eRFID[71].nCardNumber;eRFID[71].bROPPPuttedChecked;	eRFID[71].bROPPPutted;		eRFID[71].bROPPCapped;		eRFID[71].bROPPCappingAborted;eRFID[71].bROPPCappingOK; eRFID[71].bROPPCappingChecked;eRFID[71].bFormPresent; eRFID[71].bBottlePresent; eRFID[71].bDosingTwoPhases; eRFID[71].nDispencerNr; eRFID[71].nDispencerNrSecondPhase; eRFID[71].lrDoseVolumeSV; eRFID[71].lrDoseVolumeCV; eRFID[71].lrDoseVolumeSVSecondPhase; eRFID[71].lrDoseVolumeCVSecondPhase; eRFID[71].bDosed;	eRFID[71].bDoseAborted; eRFID[71].bWeighed; eRFID[71].lrWeightSV; eRFID[71].lrWeightCV; eRFID[71].lrWeightMeasuredCV; eRFID[71].bWeightOK; eRFID[71].bCapPutted; eRFID[71].bCapChecked; eRFID[71].bCapOK; eRFID[71].bCapGripperScrewed; eRFID[71].bCapGripperScrewAborted; eRFID[71].bBottleTransferedToExit; eRFID[71].bBottleTransferedToLabeler; eRFID[71].lrWeightDif; eRFID[71].lrMinWeightCV;eRFID[71].lrMaxWeightCV;
eRFID[72].nCardNumber;eRFID[72].bROPPPuttedChecked;	eRFID[72].bROPPPutted;		eRFID[72].bROPPCapped;		eRFID[72].bROPPCappingAborted;eRFID[72].bROPPCappingOK; eRFID[72].bROPPCappingChecked;eRFID[72].bFormPresent; eRFID[72].bBottlePresent; eRFID[72].bDosingTwoPhases; eRFID[72].nDispencerNr; eRFID[72].nDispencerNrSecondPhase; eRFID[72].lrDoseVolumeSV; eRFID[72].lrDoseVolumeCV; eRFID[72].lrDoseVolumeSVSecondPhase; eRFID[72].lrDoseVolumeCVSecondPhase; eRFID[72].bDosed;	eRFID[72].bDoseAborted; eRFID[72].bWeighed; eRFID[72].lrWeightSV; eRFID[72].lrWeightCV; eRFID[72].lrWeightMeasuredCV; eRFID[72].bWeightOK; eRFID[72].bCapPutted; eRFID[72].bCapChecked; eRFID[72].bCapOK; eRFID[72].bCapGripperScrewed; eRFID[72].bCapGripperScrewAborted; eRFID[72].bBottleTransferedToExit; eRFID[72].bBottleTransferedToLabeler; eRFID[72].lrWeightDif; eRFID[72].lrMinWeightCV;eRFID[72].lrMaxWeightCV;
eRFID[73].nCardNumber;eRFID[73].bROPPPuttedChecked;	eRFID[73].bROPPPutted;		eRFID[73].bROPPCapped;		eRFID[73].bROPPCappingAborted;eRFID[73].bROPPCappingOK; eRFID[73].bROPPCappingChecked;eRFID[73].bFormPresent; eRFID[73].bBottlePresent; eRFID[73].bDosingTwoPhases; eRFID[73].nDispencerNr; eRFID[73].nDispencerNrSecondPhase; eRFID[73].lrDoseVolumeSV; eRFID[73].lrDoseVolumeCV; eRFID[73].lrDoseVolumeSVSecondPhase; eRFID[73].lrDoseVolumeCVSecondPhase; eRFID[73].bDosed;	eRFID[73].bDoseAborted; eRFID[73].bWeighed; eRFID[73].lrWeightSV; eRFID[73].lrWeightCV; eRFID[73].lrWeightMeasuredCV; eRFID[73].bWeightOK; eRFID[73].bCapPutted; eRFID[73].bCapChecked; eRFID[73].bCapOK; eRFID[73].bCapGripperScrewed; eRFID[73].bCapGripperScrewAborted; eRFID[73].bBottleTransferedToExit; eRFID[73].bBottleTransferedToLabeler; eRFID[73].lrWeightDif; eRFID[73].lrMinWeightCV;eRFID[73].lrMaxWeightCV;
eRFID[74].nCardNumber;eRFID[74].bROPPPuttedChecked;	eRFID[74].bROPPPutted;		eRFID[74].bROPPCapped;		eRFID[74].bROPPCappingAborted;eRFID[74].bROPPCappingOK; eRFID[74].bROPPCappingChecked;eRFID[74].bFormPresent; eRFID[74].bBottlePresent; eRFID[74].bDosingTwoPhases; eRFID[74].nDispencerNr; eRFID[74].nDispencerNrSecondPhase; eRFID[74].lrDoseVolumeSV; eRFID[74].lrDoseVolumeCV; eRFID[74].lrDoseVolumeSVSecondPhase; eRFID[74].lrDoseVolumeCVSecondPhase; eRFID[74].bDosed;	eRFID[74].bDoseAborted; eRFID[74].bWeighed; eRFID[74].lrWeightSV; eRFID[74].lrWeightCV; eRFID[74].lrWeightMeasuredCV; eRFID[74].bWeightOK; eRFID[74].bCapPutted; eRFID[74].bCapChecked; eRFID[74].bCapOK; eRFID[74].bCapGripperScrewed; eRFID[74].bCapGripperScrewAborted; eRFID[74].bBottleTransferedToExit; eRFID[74].bBottleTransferedToLabeler; eRFID[74].lrWeightDif; eRFID[74].lrMinWeightCV;eRFID[74].lrMaxWeightCV;
eRFID[75].nCardNumber;eRFID[75].bROPPPuttedChecked;	eRFID[75].bROPPPutted;		eRFID[75].bROPPCapped;		eRFID[75].bROPPCappingAborted;eRFID[75].bROPPCappingOK; eRFID[75].bROPPCappingChecked;eRFID[75].bFormPresent; eRFID[75].bBottlePresent; eRFID[75].bDosingTwoPhases; eRFID[75].nDispencerNr; eRFID[75].nDispencerNrSecondPhase; eRFID[75].lrDoseVolumeSV; eRFID[75].lrDoseVolumeCV; eRFID[75].lrDoseVolumeSVSecondPhase; eRFID[75].lrDoseVolumeCVSecondPhase; eRFID[75].bDosed;	eRFID[75].bDoseAborted; eRFID[75].bWeighed; eRFID[75].lrWeightSV; eRFID[75].lrWeightCV; eRFID[75].lrWeightMeasuredCV; eRFID[75].bWeightOK; eRFID[75].bCapPutted; eRFID[75].bCapChecked; eRFID[75].bCapOK; eRFID[75].bCapGripperScrewed; eRFID[75].bCapGripperScrewAborted; eRFID[75].bBottleTransferedToExit; eRFID[75].bBottleTransferedToLabeler; eRFID[75].lrWeightDif; eRFID[75].lrMinWeightCV;eRFID[75].lrMaxWeightCV;
eRFID[76].nCardNumber;eRFID[76].bROPPPuttedChecked;	eRFID[76].bROPPPutted;		eRFID[76].bROPPCapped;		eRFID[76].bROPPCappingAborted;eRFID[76].bROPPCappingOK; eRFID[76].bROPPCappingChecked;eRFID[76].bFormPresent; eRFID[76].bBottlePresent; eRFID[76].bDosingTwoPhases; eRFID[76].nDispencerNr; eRFID[76].nDispencerNrSecondPhase; eRFID[76].lrDoseVolumeSV; eRFID[76].lrDoseVolumeCV; eRFID[76].lrDoseVolumeSVSecondPhase; eRFID[76].lrDoseVolumeCVSecondPhase; eRFID[76].bDosed;	eRFID[76].bDoseAborted; eRFID[76].bWeighed; eRFID[76].lrWeightSV; eRFID[76].lrWeightCV; eRFID[76].lrWeightMeasuredCV; eRFID[76].bWeightOK; eRFID[76].bCapPutted; eRFID[76].bCapChecked; eRFID[76].bCapOK; eRFID[76].bCapGripperScrewed; eRFID[76].bCapGripperScrewAborted; eRFID[76].bBottleTransferedToExit; eRFID[76].bBottleTransferedToLabeler; eRFID[76].lrWeightDif; eRFID[76].lrMinWeightCV;eRFID[76].lrMaxWeightCV;
eRFID[77].nCardNumber;eRFID[77].bROPPPuttedChecked;	eRFID[77].bROPPPutted;		eRFID[77].bROPPCapped;		eRFID[77].bROPPCappingAborted;eRFID[77].bROPPCappingOK; eRFID[77].bROPPCappingChecked;eRFID[77].bFormPresent; eRFID[77].bBottlePresent; eRFID[77].bDosingTwoPhases; eRFID[77].nDispencerNr; eRFID[77].nDispencerNrSecondPhase; eRFID[77].lrDoseVolumeSV; eRFID[77].lrDoseVolumeCV; eRFID[77].lrDoseVolumeSVSecondPhase; eRFID[77].lrDoseVolumeCVSecondPhase; eRFID[77].bDosed;	eRFID[77].bDoseAborted; eRFID[77].bWeighed; eRFID[77].lrWeightSV; eRFID[77].lrWeightCV; eRFID[77].lrWeightMeasuredCV; eRFID[77].bWeightOK; eRFID[77].bCapPutted; eRFID[77].bCapChecked; eRFID[77].bCapOK; eRFID[77].bCapGripperScrewed; eRFID[77].bCapGripperScrewAborted; eRFID[77].bBottleTransferedToExit; eRFID[77].bBottleTransferedToLabeler; eRFID[77].lrWeightDif; eRFID[77].lrMinWeightCV;eRFID[77].lrMaxWeightCV;
eRFID[78].nCardNumber;eRFID[78].bROPPPuttedChecked;	eRFID[78].bROPPPutted;		eRFID[78].bROPPCapped;		eRFID[78].bROPPCappingAborted;eRFID[78].bROPPCappingOK; eRFID[78].bROPPCappingChecked;eRFID[78].bFormPresent; eRFID[78].bBottlePresent; eRFID[78].bDosingTwoPhases; eRFID[78].nDispencerNr; eRFID[78].nDispencerNrSecondPhase; eRFID[78].lrDoseVolumeSV; eRFID[78].lrDoseVolumeCV; eRFID[78].lrDoseVolumeSVSecondPhase; eRFID[78].lrDoseVolumeCVSecondPhase; eRFID[78].bDosed;	eRFID[78].bDoseAborted; eRFID[78].bWeighed; eRFID[78].lrWeightSV; eRFID[78].lrWeightCV; eRFID[78].lrWeightMeasuredCV; eRFID[78].bWeightOK; eRFID[78].bCapPutted; eRFID[78].bCapChecked; eRFID[78].bCapOK; eRFID[78].bCapGripperScrewed; eRFID[78].bCapGripperScrewAborted; eRFID[78].bBottleTransferedToExit; eRFID[78].bBottleTransferedToLabeler; eRFID[78].lrWeightDif; eRFID[78].lrMinWeightCV;eRFID[78].lrMaxWeightCV;
eRFID[79].nCardNumber;eRFID[79].bROPPPuttedChecked;	eRFID[79].bROPPPutted;		eRFID[79].bROPPCapped;		eRFID[79].bROPPCappingAborted;eRFID[79].bROPPCappingOK; eRFID[79].bROPPCappingChecked;eRFID[79].bFormPresent; eRFID[79].bBottlePresent; eRFID[79].bDosingTwoPhases; eRFID[79].nDispencerNr; eRFID[79].nDispencerNrSecondPhase; eRFID[79].lrDoseVolumeSV; eRFID[79].lrDoseVolumeCV; eRFID[79].lrDoseVolumeSVSecondPhase; eRFID[79].lrDoseVolumeCVSecondPhase; eRFID[79].bDosed;	eRFID[79].bDoseAborted; eRFID[79].bWeighed; eRFID[79].lrWeightSV; eRFID[79].lrWeightCV; eRFID[79].lrWeightMeasuredCV; eRFID[79].bWeightOK; eRFID[79].bCapPutted; eRFID[79].bCapChecked; eRFID[79].bCapOK; eRFID[79].bCapGripperScrewed; eRFID[79].bCapGripperScrewAborted; eRFID[79].bBottleTransferedToExit; eRFID[79].bBottleTransferedToLabeler; eRFID[79].lrWeightDif; eRFID[79].lrMinWeightCV;eRFID[79].lrMaxWeightCV;
eRFID[80].nCardNumber;eRFID[80].bROPPPuttedChecked;	eRFID[80].bROPPPutted;		eRFID[80].bROPPCapped;		eRFID[80].bROPPCappingAborted;eRFID[80].bROPPCappingOK; eRFID[80].bROPPCappingChecked;eRFID[80].bFormPresent; eRFID[80].bBottlePresent; eRFID[80].bDosingTwoPhases; eRFID[80].nDispencerNr; eRFID[80].nDispencerNrSecondPhase; eRFID[80].lrDoseVolumeSV; eRFID[80].lrDoseVolumeCV; eRFID[80].lrDoseVolumeSVSecondPhase; eRFID[80].lrDoseVolumeCVSecondPhase; eRFID[80].bDosed;	eRFID[80].bDoseAborted; eRFID[80].bWeighed; eRFID[80].lrWeightSV; eRFID[80].lrWeightCV; eRFID[80].lrWeightMeasuredCV; eRFID[80].bWeightOK; eRFID[80].bCapPutted; eRFID[80].bCapChecked; eRFID[80].bCapOK; eRFID[80].bCapGripperScrewed; eRFID[80].bCapGripperScrewAborted; eRFID[80].bBottleTransferedToExit; eRFID[80].bBottleTransferedToLabeler; eRFID[80].lrWeightDif; eRFID[80].lrMinWeightCV;eRFID[80].lrMaxWeightCV;
eRFID[81].nCardNumber;eRFID[81].bROPPPuttedChecked;	eRFID[81].bROPPPutted;		eRFID[81].bROPPCapped;		eRFID[81].bROPPCappingAborted;eRFID[81].bROPPCappingOK; eRFID[81].bROPPCappingChecked;eRFID[81].bFormPresent; eRFID[81].bBottlePresent; eRFID[81].bDosingTwoPhases; eRFID[81].nDispencerNr; eRFID[81].nDispencerNrSecondPhase; eRFID[81].lrDoseVolumeSV; eRFID[81].lrDoseVolumeCV; eRFID[81].lrDoseVolumeSVSecondPhase; eRFID[81].lrDoseVolumeCVSecondPhase; eRFID[81].bDosed;	eRFID[81].bDoseAborted; eRFID[81].bWeighed; eRFID[81].lrWeightSV; eRFID[81].lrWeightCV; eRFID[81].lrWeightMeasuredCV; eRFID[81].bWeightOK; eRFID[81].bCapPutted; eRFID[81].bCapChecked; eRFID[81].bCapOK; eRFID[81].bCapGripperScrewed; eRFID[81].bCapGripperScrewAborted; eRFID[81].bBottleTransferedToExit; eRFID[81].bBottleTransferedToLabeler; eRFID[81].lrWeightDif; eRFID[81].lrMinWeightCV;eRFID[81].lrMaxWeightCV;
eRFID[82].nCardNumber;eRFID[82].bROPPPuttedChecked;	eRFID[82].bROPPPutted;		eRFID[82].bROPPCapped;		eRFID[82].bROPPCappingAborted;eRFID[82].bROPPCappingOK; eRFID[82].bROPPCappingChecked;eRFID[82].bFormPresent; eRFID[82].bBottlePresent; eRFID[82].bDosingTwoPhases; eRFID[82].nDispencerNr; eRFID[82].nDispencerNrSecondPhase; eRFID[82].lrDoseVolumeSV; eRFID[82].lrDoseVolumeCV; eRFID[82].lrDoseVolumeSVSecondPhase; eRFID[82].lrDoseVolumeCVSecondPhase; eRFID[82].bDosed;	eRFID[82].bDoseAborted; eRFID[82].bWeighed; eRFID[82].lrWeightSV; eRFID[82].lrWeightCV; eRFID[82].lrWeightMeasuredCV; eRFID[82].bWeightOK; eRFID[82].bCapPutted; eRFID[82].bCapChecked; eRFID[82].bCapOK; eRFID[82].bCapGripperScrewed; eRFID[82].bCapGripperScrewAborted; eRFID[82].bBottleTransferedToExit; eRFID[82].bBottleTransferedToLabeler; eRFID[82].lrWeightDif; eRFID[82].lrMinWeightCV;eRFID[82].lrMaxWeightCV;
eRFID[83].nCardNumber;eRFID[83].bROPPPuttedChecked;	eRFID[83].bROPPPutted;		eRFID[83].bROPPCapped;		eRFID[83].bROPPCappingAborted;eRFID[83].bROPPCappingOK; eRFID[83].bROPPCappingChecked;eRFID[83].bFormPresent; eRFID[83].bBottlePresent; eRFID[83].bDosingTwoPhases; eRFID[83].nDispencerNr; eRFID[83].nDispencerNrSecondPhase; eRFID[83].lrDoseVolumeSV; eRFID[83].lrDoseVolumeCV; eRFID[83].lrDoseVolumeSVSecondPhase; eRFID[83].lrDoseVolumeCVSecondPhase; eRFID[83].bDosed;	eRFID[83].bDoseAborted; eRFID[83].bWeighed; eRFID[83].lrWeightSV; eRFID[83].lrWeightCV; eRFID[83].lrWeightMeasuredCV; eRFID[83].bWeightOK; eRFID[83].bCapPutted; eRFID[83].bCapChecked; eRFID[83].bCapOK; eRFID[83].bCapGripperScrewed; eRFID[83].bCapGripperScrewAborted; eRFID[83].bBottleTransferedToExit; eRFID[83].bBottleTransferedToLabeler; eRFID[83].lrWeightDif; eRFID[83].lrMinWeightCV;eRFID[83].lrMaxWeightCV;
eRFID[84].nCardNumber;eRFID[84].bROPPPuttedChecked;	eRFID[84].bROPPPutted;		eRFID[84].bROPPCapped;		eRFID[84].bROPPCappingAborted;eRFID[84].bROPPCappingOK; eRFID[84].bROPPCappingChecked;eRFID[84].bFormPresent; eRFID[84].bBottlePresent; eRFID[84].bDosingTwoPhases; eRFID[84].nDispencerNr; eRFID[84].nDispencerNrSecondPhase; eRFID[84].lrDoseVolumeSV; eRFID[84].lrDoseVolumeCV; eRFID[84].lrDoseVolumeSVSecondPhase; eRFID[84].lrDoseVolumeCVSecondPhase; eRFID[84].bDosed;	eRFID[84].bDoseAborted; eRFID[84].bWeighed; eRFID[84].lrWeightSV; eRFID[84].lrWeightCV; eRFID[84].lrWeightMeasuredCV; eRFID[84].bWeightOK; eRFID[84].bCapPutted; eRFID[84].bCapChecked; eRFID[84].bCapOK; eRFID[84].bCapGripperScrewed; eRFID[84].bCapGripperScrewAborted; eRFID[84].bBottleTransferedToExit; eRFID[84].bBottleTransferedToLabeler; eRFID[84].lrWeightDif; eRFID[84].lrMinWeightCV;eRFID[84].lrMaxWeightCV;
eRFID[85].nCardNumber;eRFID[85].bROPPPuttedChecked;	eRFID[85].bROPPPutted;		eRFID[85].bROPPCapped;		eRFID[85].bROPPCappingAborted;eRFID[85].bROPPCappingOK; eRFID[85].bROPPCappingChecked;eRFID[85].bFormPresent; eRFID[85].bBottlePresent; eRFID[85].bDosingTwoPhases; eRFID[85].nDispencerNr; eRFID[85].nDispencerNrSecondPhase; eRFID[85].lrDoseVolumeSV; eRFID[85].lrDoseVolumeCV; eRFID[85].lrDoseVolumeSVSecondPhase; eRFID[85].lrDoseVolumeCVSecondPhase; eRFID[85].bDosed;	eRFID[85].bDoseAborted; eRFID[85].bWeighed; eRFID[85].lrWeightSV; eRFID[85].lrWeightCV; eRFID[85].lrWeightMeasuredCV; eRFID[85].bWeightOK; eRFID[85].bCapPutted; eRFID[85].bCapChecked; eRFID[85].bCapOK; eRFID[85].bCapGripperScrewed; eRFID[85].bCapGripperScrewAborted; eRFID[85].bBottleTransferedToExit; eRFID[85].bBottleTransferedToLabeler; eRFID[85].lrWeightDif; eRFID[85].lrMinWeightCV;eRFID[85].lrMaxWeightCV;
eRFID[86].nCardNumber;eRFID[86].bROPPPuttedChecked;	eRFID[86].bROPPPutted;		eRFID[86].bROPPCapped;		eRFID[86].bROPPCappingAborted;eRFID[86].bROPPCappingOK; eRFID[86].bROPPCappingChecked;eRFID[86].bFormPresent; eRFID[86].bBottlePresent; eRFID[86].bDosingTwoPhases; eRFID[86].nDispencerNr; eRFID[86].nDispencerNrSecondPhase; eRFID[86].lrDoseVolumeSV; eRFID[86].lrDoseVolumeCV; eRFID[86].lrDoseVolumeSVSecondPhase; eRFID[86].lrDoseVolumeCVSecondPhase; eRFID[86].bDosed;	eRFID[86].bDoseAborted; eRFID[86].bWeighed; eRFID[86].lrWeightSV; eRFID[86].lrWeightCV; eRFID[86].lrWeightMeasuredCV; eRFID[86].bWeightOK; eRFID[86].bCapPutted; eRFID[86].bCapChecked; eRFID[86].bCapOK; eRFID[86].bCapGripperScrewed; eRFID[86].bCapGripperScrewAborted; eRFID[86].bBottleTransferedToExit; eRFID[86].bBottleTransferedToLabeler; eRFID[86].lrWeightDif; eRFID[86].lrMinWeightCV;eRFID[86].lrMaxWeightCV;
eRFID[87].nCardNumber;eRFID[87].bROPPPuttedChecked;	eRFID[87].bROPPPutted;		eRFID[87].bROPPCapped;		eRFID[87].bROPPCappingAborted;eRFID[87].bROPPCappingOK; eRFID[87].bROPPCappingChecked;eRFID[87].bFormPresent; eRFID[87].bBottlePresent; eRFID[87].bDosingTwoPhases; eRFID[87].nDispencerNr; eRFID[87].nDispencerNrSecondPhase; eRFID[87].lrDoseVolumeSV; eRFID[87].lrDoseVolumeCV; eRFID[87].lrDoseVolumeSVSecondPhase; eRFID[87].lrDoseVolumeCVSecondPhase; eRFID[87].bDosed;	eRFID[87].bDoseAborted; eRFID[87].bWeighed; eRFID[87].lrWeightSV; eRFID[87].lrWeightCV; eRFID[87].lrWeightMeasuredCV; eRFID[87].bWeightOK; eRFID[87].bCapPutted; eRFID[87].bCapChecked; eRFID[87].bCapOK; eRFID[87].bCapGripperScrewed; eRFID[87].bCapGripperScrewAborted; eRFID[87].bBottleTransferedToExit; eRFID[87].bBottleTransferedToLabeler; eRFID[87].lrWeightDif; eRFID[87].lrMinWeightCV;eRFID[87].lrMaxWeightCV;
eRFID[88].nCardNumber;eRFID[88].bROPPPuttedChecked;	eRFID[88].bROPPPutted;		eRFID[88].bROPPCapped;		eRFID[88].bROPPCappingAborted;eRFID[88].bROPPCappingOK; eRFID[88].bROPPCappingChecked;eRFID[88].bFormPresent; eRFID[88].bBottlePresent; eRFID[88].bDosingTwoPhases; eRFID[88].nDispencerNr; eRFID[88].nDispencerNrSecondPhase; eRFID[88].lrDoseVolumeSV; eRFID[88].lrDoseVolumeCV; eRFID[88].lrDoseVolumeSVSecondPhase; eRFID[88].lrDoseVolumeCVSecondPhase; eRFID[88].bDosed;	eRFID[88].bDoseAborted; eRFID[88].bWeighed; eRFID[88].lrWeightSV; eRFID[88].lrWeightCV; eRFID[88].lrWeightMeasuredCV; eRFID[88].bWeightOK; eRFID[88].bCapPutted; eRFID[88].bCapChecked; eRFID[88].bCapOK; eRFID[88].bCapGripperScrewed; eRFID[88].bCapGripperScrewAborted; eRFID[88].bBottleTransferedToExit; eRFID[88].bBottleTransferedToLabeler; eRFID[88].lrWeightDif; eRFID[88].lrMinWeightCV;eRFID[88].lrMaxWeightCV;
eRFID[89].nCardNumber;eRFID[89].bROPPPuttedChecked;	eRFID[89].bROPPPutted;		eRFID[89].bROPPCapped;		eRFID[89].bROPPCappingAborted;eRFID[89].bROPPCappingOK; eRFID[89].bROPPCappingChecked;eRFID[89].bFormPresent; eRFID[89].bBottlePresent; eRFID[89].bDosingTwoPhases; eRFID[89].nDispencerNr; eRFID[89].nDispencerNrSecondPhase; eRFID[89].lrDoseVolumeSV; eRFID[89].lrDoseVolumeCV; eRFID[89].lrDoseVolumeSVSecondPhase; eRFID[89].lrDoseVolumeCVSecondPhase; eRFID[89].bDosed;	eRFID[89].bDoseAborted; eRFID[89].bWeighed; eRFID[89].lrWeightSV; eRFID[89].lrWeightCV; eRFID[89].lrWeightMeasuredCV; eRFID[89].bWeightOK; eRFID[89].bCapPutted; eRFID[89].bCapChecked; eRFID[89].bCapOK; eRFID[89].bCapGripperScrewed; eRFID[89].bCapGripperScrewAborted; eRFID[89].bBottleTransferedToExit; eRFID[89].bBottleTransferedToLabeler; eRFID[89].lrWeightDif; eRFID[89].lrMinWeightCV;eRFID[89].lrMaxWeightCV;
eRFID[90].nCardNumber;eRFID[90].bROPPPuttedChecked;	eRFID[90].bROPPPutted;		eRFID[90].bROPPCapped;		eRFID[90].bROPPCappingAborted;eRFID[90].bROPPCappingOK; eRFID[90].bROPPCappingChecked;eRFID[90].bFormPresent; eRFID[90].bBottlePresent; eRFID[90].bDosingTwoPhases; eRFID[90].nDispencerNr; eRFID[90].nDispencerNrSecondPhase; eRFID[90].lrDoseVolumeSV; eRFID[90].lrDoseVolumeCV; eRFID[90].lrDoseVolumeSVSecondPhase; eRFID[90].lrDoseVolumeCVSecondPhase; eRFID[90].bDosed;	eRFID[90].bDoseAborted; eRFID[90].bWeighed; eRFID[90].lrWeightSV; eRFID[90].lrWeightCV; eRFID[90].lrWeightMeasuredCV; eRFID[90].bWeightOK; eRFID[90].bCapPutted; eRFID[90].bCapChecked; eRFID[90].bCapOK; eRFID[90].bCapGripperScrewed; eRFID[90].bCapGripperScrewAborted; eRFID[90].bBottleTransferedToExit; eRFID[90].bBottleTransferedToLabeler; eRFID[90].lrWeightDif; eRFID[90].lrMinWeightCV;eRFID[90].lrMaxWeightCV;
eRFID[91].nCardNumber;eRFID[91].bROPPPuttedChecked;	eRFID[91].bROPPPutted;		eRFID[91].bROPPCapped;		eRFID[91].bROPPCappingAborted;eRFID[91].bROPPCappingOK; eRFID[91].bROPPCappingChecked;eRFID[91].bFormPresent; eRFID[91].bBottlePresent; eRFID[91].bDosingTwoPhases; eRFID[91].nDispencerNr; eRFID[91].nDispencerNrSecondPhase; eRFID[91].lrDoseVolumeSV; eRFID[91].lrDoseVolumeCV; eRFID[91].lrDoseVolumeSVSecondPhase; eRFID[91].lrDoseVolumeCVSecondPhase; eRFID[91].bDosed;	eRFID[91].bDoseAborted; eRFID[91].bWeighed; eRFID[91].lrWeightSV; eRFID[91].lrWeightCV; eRFID[91].lrWeightMeasuredCV; eRFID[91].bWeightOK; eRFID[91].bCapPutted; eRFID[91].bCapChecked; eRFID[91].bCapOK; eRFID[91].bCapGripperScrewed; eRFID[91].bCapGripperScrewAborted; eRFID[91].bBottleTransferedToExit; eRFID[91].bBottleTransferedToLabeler; eRFID[91].lrWeightDif; eRFID[91].lrMinWeightCV;eRFID[91].lrMaxWeightCV;
eRFID[92].nCardNumber;eRFID[92].bROPPPuttedChecked;	eRFID[92].bROPPPutted;		eRFID[92].bROPPCapped;		eRFID[92].bROPPCappingAborted;eRFID[92].bROPPCappingOK; eRFID[92].bROPPCappingChecked;eRFID[92].bFormPresent; eRFID[92].bBottlePresent; eRFID[92].bDosingTwoPhases; eRFID[92].nDispencerNr; eRFID[92].nDispencerNrSecondPhase; eRFID[92].lrDoseVolumeSV; eRFID[92].lrDoseVolumeCV; eRFID[92].lrDoseVolumeSVSecondPhase; eRFID[92].lrDoseVolumeCVSecondPhase; eRFID[92].bDosed;	eRFID[92].bDoseAborted; eRFID[92].bWeighed; eRFID[92].lrWeightSV; eRFID[92].lrWeightCV; eRFID[92].lrWeightMeasuredCV; eRFID[92].bWeightOK; eRFID[92].bCapPutted; eRFID[92].bCapChecked; eRFID[92].bCapOK; eRFID[92].bCapGripperScrewed; eRFID[92].bCapGripperScrewAborted; eRFID[92].bBottleTransferedToExit; eRFID[92].bBottleTransferedToLabeler; eRFID[92].lrWeightDif; eRFID[92].lrMinWeightCV;eRFID[92].lrMaxWeightCV;
eRFID[93].nCardNumber;eRFID[93].bROPPPuttedChecked;	eRFID[93].bROPPPutted;		eRFID[93].bROPPCapped;		eRFID[93].bROPPCappingAborted;eRFID[93].bROPPCappingOK; eRFID[93].bROPPCappingChecked;eRFID[93].bFormPresent; eRFID[93].bBottlePresent; eRFID[93].bDosingTwoPhases; eRFID[93].nDispencerNr; eRFID[93].nDispencerNrSecondPhase; eRFID[93].lrDoseVolumeSV; eRFID[93].lrDoseVolumeCV; eRFID[93].lrDoseVolumeSVSecondPhase; eRFID[93].lrDoseVolumeCVSecondPhase; eRFID[93].bDosed;	eRFID[93].bDoseAborted; eRFID[93].bWeighed; eRFID[93].lrWeightSV; eRFID[93].lrWeightCV; eRFID[93].lrWeightMeasuredCV; eRFID[93].bWeightOK; eRFID[93].bCapPutted; eRFID[93].bCapChecked; eRFID[93].bCapOK; eRFID[93].bCapGripperScrewed; eRFID[93].bCapGripperScrewAborted; eRFID[93].bBottleTransferedToExit; eRFID[93].bBottleTransferedToLabeler; eRFID[93].lrWeightDif; eRFID[93].lrMinWeightCV;eRFID[93].lrMaxWeightCV;
eRFID[94].nCardNumber;eRFID[94].bROPPPuttedChecked;	eRFID[94].bROPPPutted;		eRFID[94].bROPPCapped;		eRFID[94].bROPPCappingAborted;eRFID[94].bROPPCappingOK; eRFID[94].bROPPCappingChecked;eRFID[94].bFormPresent; eRFID[94].bBottlePresent; eRFID[94].bDosingTwoPhases; eRFID[94].nDispencerNr; eRFID[94].nDispencerNrSecondPhase; eRFID[94].lrDoseVolumeSV; eRFID[94].lrDoseVolumeCV; eRFID[94].lrDoseVolumeSVSecondPhase; eRFID[94].lrDoseVolumeCVSecondPhase; eRFID[94].bDosed;	eRFID[94].bDoseAborted; eRFID[94].bWeighed; eRFID[94].lrWeightSV; eRFID[94].lrWeightCV; eRFID[94].lrWeightMeasuredCV; eRFID[94].bWeightOK; eRFID[94].bCapPutted; eRFID[94].bCapChecked; eRFID[94].bCapOK; eRFID[94].bCapGripperScrewed; eRFID[94].bCapGripperScrewAborted; eRFID[94].bBottleTransferedToExit; eRFID[94].bBottleTransferedToLabeler; eRFID[94].lrWeightDif; eRFID[94].lrMinWeightCV;eRFID[94].lrMaxWeightCV;
eRFID[95].nCardNumber;eRFID[95].bROPPPuttedChecked;	eRFID[95].bROPPPutted;		eRFID[95].bROPPCapped;		eRFID[95].bROPPCappingAborted;eRFID[95].bROPPCappingOK; eRFID[95].bROPPCappingChecked;eRFID[95].bFormPresent; eRFID[95].bBottlePresent; eRFID[95].bDosingTwoPhases; eRFID[95].nDispencerNr; eRFID[95].nDispencerNrSecondPhase; eRFID[95].lrDoseVolumeSV; eRFID[95].lrDoseVolumeCV; eRFID[95].lrDoseVolumeSVSecondPhase; eRFID[95].lrDoseVolumeCVSecondPhase; eRFID[95].bDosed;	eRFID[95].bDoseAborted; eRFID[95].bWeighed; eRFID[95].lrWeightSV; eRFID[95].lrWeightCV; eRFID[95].lrWeightMeasuredCV; eRFID[95].bWeightOK; eRFID[95].bCapPutted; eRFID[95].bCapChecked; eRFID[95].bCapOK; eRFID[95].bCapGripperScrewed; eRFID[95].bCapGripperScrewAborted; eRFID[95].bBottleTransferedToExit; eRFID[95].bBottleTransferedToLabeler; eRFID[95].lrWeightDif; eRFID[95].lrMinWeightCV;eRFID[95].lrMaxWeightCV;
eRFID[96].nCardNumber;eRFID[96].bROPPPuttedChecked;	eRFID[96].bROPPPutted;		eRFID[96].bROPPCapped;		eRFID[96].bROPPCappingAborted;eRFID[96].bROPPCappingOK; eRFID[96].bROPPCappingChecked;eRFID[96].bFormPresent; eRFID[96].bBottlePresent; eRFID[96].bDosingTwoPhases; eRFID[96].nDispencerNr; eRFID[96].nDispencerNrSecondPhase; eRFID[96].lrDoseVolumeSV; eRFID[96].lrDoseVolumeCV; eRFID[96].lrDoseVolumeSVSecondPhase; eRFID[96].lrDoseVolumeCVSecondPhase; eRFID[96].bDosed;	eRFID[96].bDoseAborted; eRFID[96].bWeighed; eRFID[96].lrWeightSV; eRFID[96].lrWeightCV; eRFID[96].lrWeightMeasuredCV; eRFID[96].bWeightOK; eRFID[96].bCapPutted; eRFID[96].bCapChecked; eRFID[96].bCapOK; eRFID[96].bCapGripperScrewed; eRFID[96].bCapGripperScrewAborted; eRFID[96].bBottleTransferedToExit; eRFID[96].bBottleTransferedToLabeler; eRFID[96].lrWeightDif; eRFID[96].lrMinWeightCV;eRFID[96].lrMaxWeightCV;
eRFID[97].nCardNumber;eRFID[97].bROPPPuttedChecked;	eRFID[97].bROPPPutted;		eRFID[97].bROPPCapped;		eRFID[97].bROPPCappingAborted;eRFID[97].bROPPCappingOK; eRFID[97].bROPPCappingChecked;eRFID[97].bFormPresent; eRFID[97].bBottlePresent; eRFID[97].bDosingTwoPhases; eRFID[97].nDispencerNr; eRFID[97].nDispencerNrSecondPhase; eRFID[97].lrDoseVolumeSV; eRFID[97].lrDoseVolumeCV; eRFID[97].lrDoseVolumeSVSecondPhase; eRFID[97].lrDoseVolumeCVSecondPhase; eRFID[97].bDosed;	eRFID[97].bDoseAborted; eRFID[97].bWeighed; eRFID[97].lrWeightSV; eRFID[97].lrWeightCV; eRFID[97].lrWeightMeasuredCV; eRFID[97].bWeightOK; eRFID[97].bCapPutted; eRFID[97].bCapChecked; eRFID[97].bCapOK; eRFID[97].bCapGripperScrewed; eRFID[97].bCapGripperScrewAborted; eRFID[97].bBottleTransferedToExit; eRFID[97].bBottleTransferedToLabeler; eRFID[97].lrWeightDif; eRFID[97].lrMinWeightCV;eRFID[97].lrMaxWeightCV;
eRFID[98].nCardNumber;eRFID[98].bROPPPuttedChecked;	eRFID[98].bROPPPutted;		eRFID[98].bROPPCapped;		eRFID[98].bROPPCappingAborted;eRFID[98].bROPPCappingOK; eRFID[98].bROPPCappingChecked;eRFID[98].bFormPresent; eRFID[98].bBottlePresent; eRFID[98].bDosingTwoPhases; eRFID[98].nDispencerNr; eRFID[98].nDispencerNrSecondPhase; eRFID[98].lrDoseVolumeSV; eRFID[98].lrDoseVolumeCV; eRFID[98].lrDoseVolumeSVSecondPhase; eRFID[98].lrDoseVolumeCVSecondPhase; eRFID[98].bDosed;	eRFID[98].bDoseAborted; eRFID[98].bWeighed; eRFID[98].lrWeightSV; eRFID[98].lrWeightCV; eRFID[98].lrWeightMeasuredCV; eRFID[98].bWeightOK; eRFID[98].bCapPutted; eRFID[98].bCapChecked; eRFID[98].bCapOK; eRFID[98].bCapGripperScrewed; eRFID[98].bCapGripperScrewAborted; eRFID[98].bBottleTransferedToExit; eRFID[98].bBottleTransferedToLabeler; eRFID[98].lrWeightDif; eRFID[98].lrMinWeightCV;eRFID[98].lrMaxWeightCV;
eRFID[99].nCardNumber;eRFID[99].bROPPPuttedChecked;	eRFID[99].bROPPPutted;		eRFID[99].bROPPCapped;		eRFID[99].bROPPCappingAborted;eRFID[99].bROPPCappingOK; eRFID[99].bROPPCappingChecked;eRFID[99].bFormPresent; eRFID[99].bBottlePresent; eRFID[99].bDosingTwoPhases; eRFID[99].nDispencerNr; eRFID[99].nDispencerNrSecondPhase; eRFID[99].lrDoseVolumeSV; eRFID[99].lrDoseVolumeCV; eRFID[99].lrDoseVolumeSVSecondPhase; eRFID[99].lrDoseVolumeCVSecondPhase; eRFID[99].bDosed;	eRFID[99].bDoseAborted; eRFID[99].bWeighed; eRFID[99].lrWeightSV; eRFID[99].lrWeightCV; eRFID[99].lrWeightMeasuredCV; eRFID[99].bWeightOK; eRFID[99].bCapPutted; eRFID[99].bCapChecked; eRFID[99].bCapOK; eRFID[99].bCapGripperScrewed; eRFID[99].bCapGripperScrewAborted; eRFID[99].bBottleTransferedToExit; eRFID[99].bBottleTransferedToLabeler; eRFID[99].lrWeightDif; eRFID[99].lrMinWeightCV;eRFID[99].lrMaxWeightCV;
eRFID[100].nCardNumber;eRFID[100].bROPPPuttedChecked;eRFID[100].bROPPPutted;	eRFID[100].bROPPCapped;		eRFID[100].bROPPCappingAborted;eRFID[100].bROPPCappingOK;eRFID[100].bROPPCappingChecked;;eRFID[100].bFormPresent; eRFID[100].bBottlePresent; eRFID[100].bDosingTwoPhases; eRFID[100].nDispencerNr; eRFID[100].nDispencerNrSecondPhase; eRFID[100].lrDoseVolumeSV; eRFID[100].lrDoseVolumeCV; eRFID[100].lrDoseVolumeSVSecondPhase; eRFID[100].lrDoseVolumeCVSecondPhase; eRFID[100].bDoseAborted; eRFID[100].bWeighed; eRFID[100].lrWeightSV; eRFID[100].lrWeightCV; eRFID[100].lrWeightMeasuredCV; eRFID[100].bWeightOK; eRFID[100].bCapPutted; eRFID[100].bCapChecked; eRFID[100].bCapOK; eRFID[100].bCapGripperScrewed; eRFID[100].bCapGripperScrewAborted; eRFID[100].bBottleTransferedToExit; eRFID[100].bBottleTransferedToLabeler; eRFID[100].lrWeightDif; eRFID[100].lrMinWeightCV;eRFID[100].lrMinWeightCV;;
END_ACTION

ACTION aWizard:


VIS.bCapPuttedCheckSensor :=P09_CapPuttedCheck.IbCapPuttedCheckSensor;
VIS.bCapCorrectCheckCapOnSensor	:=P11_CapCorrectCheck.IbCapCorrectCheckCapOKSensor;
VIS.bCapCorrectCheckCapNotScrewedSensor :=P11_CapCorrectCheck.IbCapCorrectCheckCapNotScrewedSensor;
END_ACTION

METHOD FormDescription : STRING
VAR_INPUT
	B:BOOL;
	W:BOOL;
	N:BOOL;
	Z:BOOL;
END_VAR
IF Z THEN
	FormDescription := 'Z';
ELSIF N THEN
	FormDescription := 'N';
ELSIF W THEN
	FormDescription := 'W';
ELSIF B THEN
	FormDescription := 'B';
ELSE
	FormDescription := '';
END_IF
END_METHOD

END_PROGRAM

// ---- POUs/FB/FB_ReasonBadPackage.TcPOU
(*
Nazwa:			FB_ReasonBadPackage
Opis:			Powód odrzuceń 
Wersja:			v0.1
Data:			2019-12-17
Autor:			DP
Urzadzenia:		
Konfiguracja:	
Info: 
- 
*)
FUNCTION_BLOCK FB_ReasonBadPackage
VAR_INPUT
	bEnable: BOOL;				//Zezwolenie na pracę
	bReset:BOOL;				//Stop awaryjny nieaktywny
	tTime:TIME;					//
	bAddReason:BOOL;			//Dodaj pomiar
	bReason1:BOOL;
	sReason1Description:STRING;	//Nazwa stacji nr 1
	bReason2:BOOL;
	sReason2Description:STRING;	//Nazwa stacji nr 2
	bReason3:BOOL;
	sReason3Description:STRING;	//Nazwa stacji nr 3
	bReason4:BOOL;
	sReason4Description:STRING;	//Nazwa stacji nr 4
	bReason5:BOOL;
	sReason5Description:STRING;	//Nazwa stacji nr 5
	bReason6:BOOL;
	sReason6Description:STRING;	//Nazwa stacji nr 6
	bReason7:BOOL;
	sReason7Description:STRING;	//Nazwa stacji nr 7
	bReason8:BOOL;
	sReason8Description:STRING;	//Nazwa stacji nr 8
	bReason9:BOOL;
	sReason9Description:STRING;	//Nazwa stacji nr 9
	bReason10:BOOL;
	sReason10Description:STRING;	//Nazwa stacji nr 10
	bReason11:BOOL;
	sReason11Description:STRING;	//Nazwa stacji nr 10
	bReason12:BOOL;
	sReason12Description:STRING;	//Nazwa stacji nr 10
END_VAR

VAR_OUTPUT
	sBadPackage1:STRING;		//Opis powodu odrzuceń nr 1
	sBadPackage2:STRING;		//Opis powodu odrzuceń nr 2
	sBadPackage3:STRING;		//Opis powodu odrzuceń nr 3
	iBadPackage1:INT;			//Ilość dla powodu odrzuceń nr 1
	iBadPackage2:INT;			//Ilość dla powodu odrzuceń nr 2
	iBadPackage3:INT;			//Ilość dla powodu odrzuceń nr3
END_VAR

VAR
	arReason: ARRAY [1..12] OF S_CycleTimes;
	i: INT;
	rtAddReason: R_TRIG;
	tonResetCounters: TON;
	dTimeTempReason1: DINT;
	dTimeTempReason2: DINT;
	dTimeTempReason3: DINT;
END_VAR

ErrorHandling();
Cycle();
ManualMovements();
Statistics();

ACTION Cycle:
tonResetCounters(IN:=NOT tonResetCounters.Q, PT:=tTime); // Resetowanie liczników
tonResetCounters.ET;
IF tonResetCounters.Q THEN
	FOR i:=1 TO 12 DO
		arReason[i].dTime :=0;
	END_FOR
	sBadPackage1 := '';
	sBadPackage2 := '';
	sBadPackage3 := '';	
	iBadPackage1 := 0;
	iBadPackage2 := 0;
	iBadPackage3 := 0;	
END_IF

rtAddReason(CLK:=bAddReason,Q=>);
IF rtAddReason.Q THEN
	IF bReason1 THEN
		arReason[1].dTime := arReason[1].dTime +1 ;
	ELSIF bReason2 THEN		                
		arReason[2].dTime := arReason[2].dTime +1 ;
	ELSIF bReason3 THEN		                
		arReason[3].dTime := arReason[3].dTime +1 ;
	ELSIF bReason4 THEN		                
		arReason[4].dTime := arReason[4].dTime +1 ;
	ELSIF bReason5 THEN		                
		arReason[5].dTime := arReason[5].dTime +1 ;
	ELSIF bReason6 THEN		                
		arReason[6].dTime := arReason[6].dTime +1 ;
	ELSIF bReason7 THEN		                
		arReason[7].dTime := arReason[7].dTime +1 ;
	ELSIF bReason8 THEN		                
		arReason[8].dTime := arReason[8].dTime +1 ;
	ELSIF bReason9 THEN		                
		arReason[9].dTime := arReason[9].dTime +1 ;
	ELSIF bReason10 THEN		                
		arReason[10].dTime := arReason[10].dTime +1 ;
	ELSIF bReason11 THEN		                
		arReason[11].dTime := arReason[11].dTime +1 ;
	ELSIF bReason12 THEN		                
		arReason[12].dTime := arReason[12].dTime +1 ;
	END_IF
END_IF

dTimeTempReason1:=0;
dTimeTempReason2:=0;
dTimeTempReason3:=0;
arReason[1].bName:=sReason1Description;
arReason[2].bName:=sReason2Description;
arReason[3].bName:=sReason3Description;
arReason[4].bName:=sReason4Description;
arReason[5].bName:=sReason5Description;
arReason[6].bName:=sReason6Description;
arReason[7].bName:=sReason7Description;
arReason[8].bName:=sReason8Description;
arReason[9].bName:=sReason9Description;
arReason[10].bName:=sReason10Description;
arReason[11].bName:=sReason11Description;
arReason[12].bName:=sReason12Description;

IF rtAddReason.Q THEN

	FOR i:=1 TO 12 DO
		IF arReason[i].dTime > dTimeTempReason1 AND arReason[i].dTime > 0 THEN
			dTimeTempReason1:=arReason[i].dTime;
			//sBadPackage1:=CONCAT(arReason[i].bName,CONCAT(' : ',DINT_TO_STRING(dTimeTempReason1))); 
			sBadPackage1:=arReason[i].bName;
			iBadPackage1:=DINT_TO_INT(dTimeTempReason1);
		END_IF
	END_FOR
	
	FOR i:=1 TO 12 DO
		IF NOT (dTimeTempReason1 = arReason[i].dTime) AND arReason[i].dTime > 0 AND arReason[i].dTime > dTimeTempReason2 THEN
			dTimeTempReason2:=arReason[i].dTime;
			//sBadPackage2:=CONCAT(arReason[i].bName,CONCAT(' : ',DINT_TO_STRING(dTimeTempReason2))); 
			sBadPackage2:=arReason[i].bName;
			iBadPackage2:=DINT_TO_INT(dTimeTempReason2);
		END_IF
	END_FOR
		
	
	FOR i:=1 TO 12 DO
		IF NOT (dTimeTempReason1 = arReason[i].dTime) AND NOT (dTimeTempReason2 = arReason[i].dTime) AND arReason[i].dTime > 0 AND arReason[i].dTime > dTimeTempReason3 THEN
			dTimeTempReason3:=arReason[i].dTime;
			//sBadPackage3:=CONCAT(arReason[i].bName,CONCAT(' : ',DINT_TO_STRING(dTimeTempReason3))); 
			sBadPackage3:=arReason[i].bName;
			iBadPackage3:=DINT_TO_INT(dTimeTempReason3);
		END_IF
	END_FOR

END_IF
END_ACTION

ACTION ErrorHandling:

END_ACTION

ACTION ManualMovements:

END_ACTION

ACTION Statistics:

END_ACTION

END_FUNCTION_BLOCK

// ---- POUs/FB/FB_2ReasonBadPackageWithID.TcPOU
(*
Nazwa:			FB_ReasonBadPackage
Opis:			Powód odrzuceń 
Wersja:			v0.28
Data:			2026-01-13
Autor:			DP
Urzadzenia:		
Konfiguracja:	
Zmiany:
- 20260113[DP] Ostatni odzut wpsisany na sama górę
- 20250818 [DP] Ostatni odzut wpsisany na sama górę, jeszcze do poprawienia
- Dodany ROPP
Info: 
- 
*)
FUNCTION_BLOCK FB_2ReasonBadPackageWithID
VAR_INPUT	
	bEnable:BOOL;					//Zezwolenie na pracę
	tTime:TIME;					
	bReason1:BOOL;              	
	sReason1Description:STRING;		//Nazwa stacji nr 1
	bReason2:BOOL;              	
	sReason2Description:STRING;		//Nazwa stacji nr 2
	bReason3:BOOL;              	
	sReason3Description:STRING;		//Nazwa stacji nr 3
	bReason4:BOOL;              	
	sReason4Description:STRING;		//Nazwa stacji nr 4
	bReason5:BOOL;              	
	sReason5Description:STRING;		//Nazwa stacji nr 5
	bReason6:BOOL;              	
	sReason6Description:STRING;		//Nazwa stacji nr 6
	bReason7:BOOL;              	
	sReason7Description:STRING;		//Nazwa stacji nr 7
	bReason8:BOOL;              	
	sReason8Description:STRING;		//Nazwa stacji nr 8
	bReason9:BOOL;              	
	sReason9Description:STRING;		//Nazwa stacji nr 9
	bReason10:BOOL;             	
	sReason10Description:STRING;	//Nazwa stacji nr 10
	bReason11:BOOL;             	
	sReason11Description:STRING;	//Nazwa stacji nr 11
	bReason12:BOOL;             	
	sReason12Description:STRING;	//Nazwa stacji nr 12
	bReason13:BOOL;             	
	sReason13Description:STRING;	//Nazwa stacji nr 13
	bReason14:BOOL;             	
	sReason14Description:STRING;	//Nazwa stacji nr 14
	bReason21:BOOL;
	sReason21Description:STRING;	//Nazwa stacji nr 1
	bReason22:BOOL;
	sReason22Description:STRING;	//Nazwa stacji nr 2
	bReason23:BOOL;
	sReason23Description:STRING;	//Nazwa stacji nr 3
	bReason24:BOOL;
	sReason24Description:STRING;	//Nazwa stacji nr 4
	bReason25:BOOL;
	sReason25Description:STRING;	//Nazwa stacji nr 5
	bReason26:BOOL;
	sReason26Description:STRING;	//Nazwa stacji nr 6
	bReason27:BOOL;
	sReason27Description:STRING;	//Nazwa stacji nr 7
	bReason28:BOOL;
	sReason28Description:STRING;	//Nazwa stacji nr 8
	bReason29:BOOL;
	sReason29Description:STRING;	//Nazwa stacji nr 9
	bReason210:BOOL;
	sReason210Description:STRING;	//Nazwa stacji nr 10
	bReason211:BOOL;
	sReason211Description:STRING;	//Nazwa stacji nr 11	
	bReason212:BOOL;
	sReason212Description:STRING;	//Nazwa stacji nr 12		
	bReason213:BOOL;
	sReason213Description:STRING;	//Nazwa stacji nr 13	
	bReason214:BOOL;
	sReason214Description:STRING;	//Nazwa stacji nr 14		
END_VAR

VAR_IN_OUT
	bAddReason1:BOOL;	
	bAddReason2:BOOL;		
	bClear:BOOL;				
END_VAR

VAR_OUTPUT
	AStReason					:ARRAY[0..63] OF S_Information;
END_VAR

VAR
	i: INT;
	rtAddReason: R_TRIG;
	tonResetCounters: TON;

	bReasonNew: BOOL;
	iReason1: INT;
	iReason2: INT;
	iReason3: INT;
	iReason4: INT;
	iReason5: INT;
	iReason6: INT;
	iReason7: INT;
	iReason8: INT;
	iReason9: INT;
	iReason10: INT;
	iReason11: INT;
	iReason12: INT;
	iReason13: INT;	
	iReason14: INT;
	
	iReason21: INT;
	iReason22: INT;
	iReason23: INT;
	iReason24: INT;
	iReason25: INT;
	iReason26: INT;
	iReason27: INT;
	iReason28: INT;
	iReason29: INT;
	iReason210: INT;
	iReason211: INT;
	iReason212: INT;
	iReason213: INT;
	iReason214: INT;
	
	rtAddReason2: R_TRIG;
	n: INT;
	iNoReason1: INT;
	iNoReason2: INT;
	AStReasonTemp	: S_Information;
END_VAR

ErrorHandling();
Cycle();
ManualMovements();
Statistics();

ACTION Cycle:
//tonResetCounters(IN:=NOT tonResetCounters.Q, PT:=tTime); // Resetowanie liczników
tonResetCounters.ET;
IF tonResetCounters.Q OR bClear THEN
	FOR i:=0 TO 63 DO
		AStReason[i].udiID :=0;
		AStReason[i].wsDescription :="";		
	END_FOR
	iReason1	:=	iReason21	:= 0;
	iReason2	:=	iReason22	:= 0;
	iReason3	:=	iReason23	:= 0;
	iReason4	:=	iReason24	:= 0;
	iReason5	:=	iReason25	:= 0;
	iReason6	:=	iReason26	:= 0;
	iReason7	:=	iReason27	:= 0;
	iReason8	:=	iReason28	:= 0;
	iReason9	:=	iReason29	:= 0;
	iReason10   :=	iReason210  := 0;
	iReason11   :=	iReason211  := 0;
	iReason12   :=	iReason212  := 0;	
	iReason13   :=	iReason213  := 0;	
	iReason14   :=	iReason214  := 0;	
	
	bAddReason1	:=	FALSE;
	bAddReason2	:=	FALSE;	
	bClear	:=	FALSE;
END_IF

rtAddReason	(CLK:=	bAddReason1,	Q=>);

IF rtAddReason.Q THEN
	
	IF	 bReason1 THEN			IF M_Add(sReason1Description:=sReason1Description,AstReason:=AStReason,AstReasonTemp:=AStReasonTemp) 	THEN	bAddReason1	:=	FALSE;	END_IF	iReason1	:=	iReason1	+	1;
	ELSIF bReason2 THEN			IF M_Add(sReason1Description:=sReason2Description,AstReason:=AStReason,AstReasonTemp:=AStReasonTemp) 	THEN	bAddReason1	:=	FALSE;	END_IF	iReason2	:=	iReason2	+	1;
	ELSIF bReason3 THEN			IF M_Add(sReason1Description:=sReason3Description,AstReason:=AStReason,AstReasonTemp:=AStReasonTemp) 	THEN	bAddReason1	:=	FALSE;	END_IF	iReason3	:=	iReason3	+	1;
	ELSIF bReason4 THEN			IF M_Add(sReason1Description:=sReason4Description,AstReason:=AStReason,AstReasonTemp:=AStReasonTemp) 	THEN	bAddReason1	:=	FALSE;	END_IF	iReason4	:=	iReason4	+	1;
	ELSIF bReason5 THEN			IF M_Add(sReason1Description:=sReason5Description,AstReason:=AStReason,AstReasonTemp:=AStReasonTemp) 	THEN	bAddReason1	:=	FALSE;	END_IF	iReason5	:=	iReason5	+	1;
	ELSIF bReason6 THEN			IF M_Add(sReason1Description:=sReason6Description,AstReason:=AStReason,AstReasonTemp:=AStReasonTemp) 	THEN	bAddReason1	:=	FALSE;	END_IF	iReason6	:=	iReason6	+	1;
	ELSIF bReason7 THEN			IF M_Add(sReason1Description:=sReason7Description,AstReason:=AStReason,AstReasonTemp:=AStReasonTemp) 	THEN	bAddReason1	:=	FALSE;	END_IF	iReason7	:=	iReason7	+	1;
	ELSIF bReason8 THEN			IF M_Add(sReason1Description:=sReason8Description,AstReason:=AStReason,AstReasonTemp:=AStReasonTemp) 	THEN	bAddReason1	:=	FALSE;	END_IF	iReason8	:=	iReason8	+	1;
	ELSIF bReason9 THEN			IF M_Add(sReason1Description:=sReason9Description,AstReason:=AStReason,AstReasonTemp:=AStReasonTemp) 	THEN	bAddReason1	:=	FALSE;	END_IF	iReason9	:=	iReason9	+	1;
	ELSIF bReason10 THEN		IF M_Add(sReason1Description:=sReason10Description,AstReason:=AStReason,AstReasonTemp:=AStReasonTemp) 	THEN	bAddReason1	:=	FALSE;	END_IF	iReason10	:=	iReason10	+	1;
	ELSIF bReason11 THEN		IF M_Add(sReason1Description:=sReason11Description,AstReason:=AStReason,AstReasonTemp:=AStReasonTemp)  	THEN	bAddReason1	:=	FALSE;	END_IF	iReason11	:=	iReason11	+	1;
	ELSIF bReason12 THEN		IF M_Add(sReason1Description:=sReason12Description,AstReason:=AStReason,AstReasonTemp:=AStReasonTemp)  	THEN	bAddReason1	:=	FALSE;	END_IF	iReason12	:=	iReason12	+	1;
	ELSIF bReason13 THEN		IF M_Add(sReason1Description:=sReason13Description,AstReason:=AStReason,AstReasonTemp:=AStReasonTemp)  	THEN	bAddReason1	:=	FALSE;	END_IF	iReason13	:=	iReason13	+	1;
	ELSIF bReason14 THEN		IF M_Add(sReason1Description:=sReason14Description,AstReason:=AStReason,AstReasonTemp:=AStReasonTemp)  	THEN	bAddReason1	:=	FALSE;	END_IF	iReason14	:=	iReason14	+	1;

	ELSE
		M_Add(sReason1Description:=sReason7Description,AstReason:=AStReason,AstReasonTemp:=AStReasonTemp);//ROPP
		iNoReason1	:=	iNoReason1	+	1; bAddReason1	:=	FALSE;
	END_IF
	
	(**Sortowanie tablicy**)
	n := 63;
	WHILE n>1 DO
		FOR i := 0 TO 63-1 DO

			IF AStReason[i].udiID = 0 THEN //Jeżeli pusty
				AStReason[i].udiID				:=	AStReason[i+1].udiID;
				AStReason[i].wsDescription		:=	AStReason[i+1].wsDescription;			
				AStReason[i+1].udiID			:=	0;
				AStReason[i+1].wsDescription	:=	"";			
			END_IF		
		END_FOR
		n := n - 1;
	END_WHILE	
	
END_IF


rtAddReason2(CLK:=bAddReason2,Q=>);

IF rtAddReason2.Q THEN
	
	IF	 bReason21 THEN			IF M_Add(sReason1Description:=sReason21Description,AstReason:=AStReason,AstReasonTemp:=AStReasonTemp)  		THEN	bAddReason2	:=	FALSE;	END_IF	iReason21	:=	iReason21	+	1;
	ELSIF bReason22 THEN		IF M_Add(sReason1Description:=sReason22Description,AstReason:=AStReason,AstReasonTemp:=AStReasonTemp)  		THEN	bAddReason2	:=	FALSE;	END_IF	iReason22	:=	iReason22	+	1;
	ELSIF bReason23 THEN		IF M_Add(sReason1Description:=sReason23Description,AstReason:=AStReason,AstReasonTemp:=AStReasonTemp)  		THEN	bAddReason2	:=	FALSE;	END_IF	iReason23	:=	iReason23	+	1;
	ELSIF bReason24 THEN		IF M_Add(sReason1Description:=sReason24Description,AstReason:=AStReason,AstReasonTemp:=AStReasonTemp)  		THEN	bAddReason2	:=	FALSE;	END_IF	iReason24	:=	iReason24	+	1;
	ELSIF bReason25 THEN		IF M_Add(sReason1Description:=sReason25Description,AstReason:=AStReason,AstReasonTemp:=AStReasonTemp)  		THEN	bAddReason2	:=	FALSE;	END_IF	iReason25	:=	iReason25	+	1;
	ELSIF bReason26 THEN		IF M_Add(sReason1Description:=sReason26Description,AstReason:=AStReason,AstReasonTemp:=AStReasonTemp)  		THEN	bAddReason2	:=	FALSE;	END_IF	iReason26	:=	iReason26	+	1;
	ELSIF bReason27 THEN		IF M_Add(sReason1Description:=sReason27Description,AstReason:=AStReason,AstReasonTemp:=AStReasonTemp)  		THEN	bAddReason2	:=	FALSE;	END_IF	iReason27	:=	iReason27	+	1;
	ELSIF bReason28 THEN		IF M_Add(sReason1Description:=sReason28Description,AstReason:=AStReason,AstReasonTemp:=AStReasonTemp)  		THEN	bAddReason2	:=	FALSE;	END_IF	iReason28	:=	iReason28	+	1;
	ELSIF bReason29 THEN		IF M_Add(sReason1Description:=sReason29Description,AstReason:=AStReason,AstReasonTemp:=AStReasonTemp)  		THEN	bAddReason2	:=	FALSE;	END_IF	iReason29	:=	iReason29	+	1;
	ELSIF bReason210 THEN		IF M_Add(sReason1Description:=sReason210Description,AstReason:=AStReason,AstReasonTemp:=AStReasonTemp)  	THEN	bAddReason2	:=	FALSE;	END_IF	iReason210	:=	iReason210	+	1;
	ELSIF bReason211 THEN		IF M_Add(sReason1Description:=sReason211Description,AstReason:=AStReason,AstReasonTemp:=AStReasonTemp)  	THEN	bAddReason2	:=	FALSE;	END_IF	iReason211	:=	iReason211	+	1;
	ELSIF bReason212 THEN		IF M_Add(sReason1Description:=sReason212Description,AstReason:=AStReason,AstReasonTemp:=AStReasonTemp)  	THEN	bAddReason2	:=	FALSE;	END_IF	iReason212	:=	iReason212	+	1;
	ELSIF bReason213 THEN		IF M_Add(sReason1Description:=sReason213Description,AstReason:=AStReason,AstReasonTemp:=AStReasonTemp)  	THEN	bAddReason2	:=	FALSE;	END_IF	iReason213	:=	iReason213	+	1;
	ELSIF bReason214 THEN		IF M_Add(sReason1Description:=sReason214Description,AstReason:=AStReason,AstReasonTemp:=AStReasonTemp)  	THEN	bAddReason2	:=	FALSE;	END_IF	iReason214	:=	iReason214	+	1;

	ELSE
		M_Add(sReason1Description:=sReason27Description,AstReason:=AStReason,AstReasonTemp:=AStReasonTemp);//ROPP
		iNoReason2	:=	iNoReason2	+	1;	bAddReason2	:=	FALSE;
	END_IF

	(**Sortowanie tablicy**)
	n := 63;
	WHILE n>1 DO
		FOR i := 0 TO 63-1 DO

			IF AStReason[i].udiID = 0 THEN //Jeżeli pusty
				AStReason[i].udiID				:=	AStReason[i+1].udiID;
				AStReason[i].wsDescription		:=	AStReason[i+1].wsDescription;			
				AStReason[i+1].udiID			:=	0;
				AStReason[i+1].wsDescription	:=	"";			
			END_IF		
		END_FOR
		n := n - 1;
	END_WHILE	
	
END_IF

AStReason[0].udiID;AStReason[0].wsDescription;
AStReason[1].udiID;AStReason[1].wsDescription;
AStReason[2].udiID;AStReason[2].wsDescription;
AStReason[3].udiID;AStReason[3].wsDescription;
AStReason[4].udiID;AStReason[4].wsDescription;
AStReason[5].udiID;AStReason[5].wsDescription;
AStReason[6].udiID;AStReason[6].wsDescription;
AStReason[7].udiID;AStReason[7].wsDescription;
AStReason[8].udiID;AStReason[8].wsDescription;
AStReason[9].udiID;AStReason[9].wsDescription;
AStReason[10].udiID;AStReason[10].wsDescription;
END_ACTION

ACTION ErrorHandling:

END_ACTION



METHOD M_Add : BOOL

VAR_INPUT
	sReason1Description		:STRING;
END_VAR
VAR_IN_OUT
	AStReason				:ARRAY[0..63] OF S_Information;
	AStReasonTemp			:S_Information;		
END_VAR
VAR
	i,j: INT;
	bReasonNew: BOOL;
END_VAR
		FOR i := 0 TO 63-1 DO
			bReasonNew	:=	TRUE;
			IF AStReason[i].udiID = STRING_TO_UDINT(sReason1Description) THEN
				AStReason[i].wsDescription 	:=	UDINT_TO_WSTRING(WSTRING_TO_UDINT(AStReason[i].wsDescription)+1);
				bReasonNew					:=	FALSE;
				//DODANE
				AStReasonTemp	:=	AStReason[i];
				FOR j := 0 TO i-1 DO
					AStReason[i-j]:=AStReason[i-j-1];
				END_FOR
				AStReason[0]:= AStReasonTemp;
				//DODANE KONIEC
				//AStReason[0]	:=	AStReason[i];
				//AStReason[i]	:=  AStReasonTemp;
		
				EXIT;
			END_IF
		END_FOR
		IF bReasonNew THEN
			FOR i := 0 TO 63-1 DO
				IF AStReason[i].udiID = 0 THEN
					AStReason[i].udiID			:=	STRING_TO_UDINT(sReason1Description);
					AStReason[i].wsDescription 	:=	UDINT_TO_WSTRING(WSTRING_TO_UDINT(AStReason[i].wsDescription)+1);
					bReasonNew	:=	FALSE;
					//DODANE
					AStReasonTemp	:=	AStReason[i];
					FOR j := 0 TO i-1 DO
						AStReason[i-j]:=AStReason[i-j-1];
					END_FOR
					AStReason[0]:= AStReasonTemp;
					//DODANE KONIEC
					//AStReasonTemp	:=	AStReason[0];
					//AStReason[0]	:=	AStReason[i];
					//AStReason[i]	:=  AStReasonTemp;
					
					EXIT;
				END_IF
			END_FOR
			
		END_IF
		M_Add := TRUE;
END_METHOD

ACTION ManualMovements:

END_ACTION

ACTION Statistics:

END_ACTION

END_FUNCTION_BLOCK

// ---- POUs/FB/FB_MoveRegister.TcPOU
(*
Nazwa:			FB_MoveRegister
Opis:			Blok przesuniecia rejestru formatek
Wersja:			v0.3 		
Data:			2018-11-16
Autor:			DP
Urzadzenia:		 
Konfiguracja:	
Info:
- Są dwa rejestry, wejściowy i wyjsciowy (struktury)
- Jezeli rejestr ma np. 6 elementów to za kazdym razem po wykryciu trigera program będzie
	1 wejściowy przesuwał na 1 wolny (nie ma formatki) wyjściowy
	kasował 1 rejestr wejściowy
	przesuwal rejetr wejsciowy 2 na 1(przeniesiony i skasowany), 3 na 2, 4 na 3, 5 na 4, 6 na 5 i kasowal 6wejsciowy
	tym sposobem po 6 trigerach caly rejestr wejsciowy powinien być na wyjsciowym
	np po 3 trigerach na wyjsciowym powinny byc zajete 1 do 3 i na wejsciowym 1 do 3
Błędy:
1 - nie wyszło z pętli for
2 - formatka już jest w rejestrze
Uwagi:
- 
Zmiany:
2018-09-18 Dodano sprawdzanie nasadek
2018-06-14 DP Pierwsza wersja
*)

FUNCTION_BLOCK FB_MoveRegister
VAR_INPUT
	bFirstCycle:BOOL;					//Pierwszy cykl, zeby na początku nie wykrywało zbocza opadającego
	bTrigger :BOOL;						// Przesuniecie tablicy o jeden
	tTriggerFilterTimeOn:TIME:=T#0MS;	// Czas filtrowania wejścia Trigger na załączenie
	tTriggerFilterTimeOff:TIME:=T#0MS;	// Czas filtrowania wejścia Trigger na wyłączenie
	bTriggerBottle :BOOL;				// Zapisywanie czy jest butelka czy nie (jezeli kontrola wlączona)
	bWithBottleControl: BOOL;			// Włączona opcja kontroli butelek
	bWithCapControl:BOOL;				// Wlaczona kontrola nasadek
	bWithFormControlTrigerCounter:BOOL;	// Jezeku na trigercontrol nie ma formatki do przesunięcia to stwórz nową
	bMoveOnlyToLastExitRegister:BOOL;	// Przepisuj rejestr wejściowy tylko na ostatni wyjściowy bez przesunięcia wyjściowego
	bMoveOnlyIfFormPresent:BOOL;		// Przepisuj tylko jak jest formatka
	bRotateEntranceRegisterBefore:BOOL;	// Najpierw przesuń rejestr wejściowy a następnie z niego zabierz
	bNoKeepTryingMove:BOOL;				// Dalej przepisuj jezeli nie ma miejsca
	bTriggerCap: BOOL;					// Truger wykrycia nasadki
	bReset :BOOL;						// Czyszczenie tablic
	iEntranceArrayElements :UINT; 		// Wartość koncowa tablicy
	iExitArrayElements :UINT; 			// Wartość koncowa tablicy
	bInvertWriting :BOOL;				// Wpisywanie odwrotne zamist z 1entrance na 1exit to 1entrance na 6exit	
	eClearPackageState :S_PackageState; // Czysty rejestr
END_VAR
VAR_IN_OUT
	bTriggerCounter :BOOL;		// Triger ktory jest kasowany
	eEntranceState :ARRAY [1..17] OF S_PackageState;	
	eExitState :ARRAY [1..17] OF S_PackageState;
	bKeepTryingMove :BOOL;		// Probuj dalej zapisać formatki aż się któraś zwolni
END_VAR

VAR_OUTPUT	
	bError :BOOL; 				// Błąd
	iError: UINT;				// Nr Błędu
	bTriggerDone :BOOL; 		// Wykonano przesunięcie
	bTriggerFilteredOUT:BOOL;	//Wyjscie przefiltrowanego sygnalu wejsciowego
END_VAR

VAR
	i:UINT;						// Zmienna w tablicy
	k:UINT;						// Pomocnicza zmienna do zapisywnia czy jest butelka
	rtbTrigger :R_TRIG;			// Reaguje na zbocze
	rtbTriggerBottle :R_TRIG;	// Reaguje na zbocze
	rtbReset :R_TRIG;			// Reaguje na zbocze
	TimerResetErrors :TON;		// Reset Błedu
	nFormCounter :UINT;					//Licznik formatek
	r1,r2:UINT;
	bBottlePresent: BOOL;				//Zmienna pomocnicza ze wykryto butelkę
	bCapPresent: BOOL;					//Zmienna pomocnicza ze wykryto butelkę
	j: UINT;
	tonTriggerFilterTimeOn: TON;
	bTriggerFiltered: BOOL;
	tofTriggerFilterTimeOff: TOF;
	tonTriggerFilterTimeBeforeTrigger: TON;
END_VAR

//Filtrowanie sygnału wejściowego
tofTriggerFilterTimeOff	(IN:=bTrigger, PT:=tTriggerFilterTimeOff);
tonTriggerFilterTimeOn	(IN:=tofTriggerFilterTimeOff.Q, PT:=tTriggerFilterTimeOn);
bTriggerFiltered 		:= tonTriggerFilterTimeOn.Q;
bTriggerFilteredOUT		:= bTriggerFiltered ;

//TRIGI I TIMERY
IF bWithBottleControl THEN
	rtbTrigger 	(CLK := NOT bTriggerFiltered, Q=>);
	rtbTriggerBottle 	(CLK := NOT bTriggerBottle, Q=>);
ELSIF bWithCapControl THEN
	rtbTrigger 	(CLK := NOT bTriggerFiltered, Q=>);
ELSE
	rtbTrigger 	(CLK := bTriggerFiltered, Q=>);
	rtbTriggerBottle 	(CLK := bTriggerBottle, Q=>);
END_IF

rtbReset 	(CLK := bReset, Q=>);
TimerResetErrors (IN:= bError, PT:=T#1000MS, Q=>);

//RESETOWANIE BLEDU
IF TimerResetErrors.Q THEN
	bError := FALSE;
END_IF

//KASOWANIE ZMIENNYCH
bTriggerDone := FALSE;

//JEZELI WLACZONO KONTROLE BUTELEK TO NADPISUJ REJESTR CZY JEST BUTELKA
IF bWithBottleControl AND bTrigger AND bTriggerBottle AND NOT bKeepTryingMove THEN //Jezeli od wykrycia formatki liczy TIMER i wykryło butelke to wpisz do rejestru że jest butelka
	eEntranceState[1].bBottlePresent := TRUE;
	eEntranceState[1].bFormPresent := TRUE;
	bBottlePresent := TRUE; // Wpisuje że jest butelka jezeli wystąpi sygnał podczas trwania czujnika formatki
ELSIF bWithBottleControl AND rtbTrigger.Q AND NOT bBottlePresent AND  NOT bKeepTryingMove AND bFirstCycle THEN
	eEntranceState[1].bBottlePresent := FALSE;
	eEntranceState[1].bFormPresent := TRUE; // jeżeli zanik czujnik formatki i nie było formatki to wpisz ze nie było butelki
END_IF
//JEZELI WLACZONO KONTROLE NASADEk TO NADPISUJ REJESTR CZY JEST BUTELKA 
(*IF bWithCapControl AND bTrigger AND bTriggerCap AND NOT bKeepTryingMove THEN //Jezeli od wykrycia formatki liczy TIMER i wykryło butelke to wpisz do rejestru że jest butelka
	eEntranceState[1].bCapPutted := TRUE;
	eEntranceState[1].bCapOK := TRUE; eEntranceState[1].bBottlePresent:= TRUE;//Zmiana nowa
	eEntranceState[1].bFormPresent := TRUE;
	bCapPresent := TRUE; // Wpisuje że jest butelka jezeli wystąpi sygnał podczas trwania czujnika formatki*)
	//ZMIANA LU 192
IF bWithCapControl AND bTriggerCap AND NOT bKeepTryingMove THEN //Jezeli od wykrycia formatki liczy TIMER i wykryło butelke to wpisz do rejestru że jest butelka
	eEntranceState[1].bCapPutted := TRUE;
	eEntranceState[1].bCapOK := TRUE; eEntranceState[1].bBottlePresent:= TRUE;//Zmiana nowa
	eEntranceState[1].bFormPresent := TRUE;
	bCapPresent := TRUE; // Wpisuje że jest butelka jezeli wystąpi sygnał podczas trwania czujnika formatki	
ELSIF bWithCapControl AND rtbTrigger.Q AND NOT bCapPresent AND  NOT bKeepTryingMove AND bFirstCycle THEN
	eEntranceState[1].bCapPutted := TRUE;
	eEntranceState[1].bCapOK:= FALSE;
	eEntranceState[1].bFormPresent := TRUE; // jeżeli zanik czujnik formatki i nie było formatki to wpisz ze nie było butelki
END_IF
//JEZELI WLACZONO SPRAWDZANIE FORMATEK Z TRIGERCOUNTER TO
IF bWithFormControlTrigerCounter  AND (bTriggerCounter OR rtbTrigger.Q) AND NOT bKeepTryingMove AND bFirstCycle THEN //Zmiena UBL50, tworz tez nowa jak Trigger
	eEntranceState[1].bFormPresent := TRUE;
END_IF



//PRZESUNIECIE
IF iEntranceArrayElements = iExitArrayElements AND bFirstCycle AND NOT bMoveOnlyToLastExitRegister THEN
	IF rtbTrigger.Q OR bKeepTryingMove OR bTriggerCounter THEN
		bTriggerCounter := FALSE; 
		bKeepTryingMove := FALSE;
		nFormCounter := 0;
		bBottlePresent:= bCapPresent  := FALSE; 
		IF NOT bInvertWriting THEN // Jezeli odwrotne wpisywanie
			FOR i := 1 TO iEntranceArrayElements DO
				IF  NOT eExitState[i].bFormPresent THEN  		// Jeżeli w rejestrze wyjściowym jest wolne miejsce to wpisz rejestr wejściowy
					eExitState[i] := eEntranceState[1];	// Wpisz do rejestru dane np z [1] Buffor do [1,2,3,4,5,6] Package
					eEntranceState[1]:=eClearPackageState;	// Czyszczenie pierwszego rejestru wejściowego
					k:=i;											// Przepisywanie zmiennej pomocniczej
					FOR i := 1 TO iEntranceArrayElements DO   				
						IF i = iEntranceArrayElements THEN
							eEntranceState[i]:=eClearPackageState;		  // Zerowanie ostatniego bo zostało przesuniete wszystko o 1
						ELSE													  // Przepisanie 2 do 1, 3 do 2, 4 do 3, 5 do 4, 6 do 5, zeruj 6
							eEntranceState[i] := eEntranceState[i+1]; // 2 do 1, 3 do 2,
							eEntranceState[i+1]:=eClearPackageState;		  // zeruj 2, 
						END_IF
					END_FOR
					bTriggerDone := TRUE;
					EXIT;
					bError := TRUE;
					iError := 1;
				ELSE
					nFormCounter := nFormCounter + 1;
					bError := TRUE;
					iError := 2;
				END_IF
			END_FOR
		ELSE
		
		//jezeli wybrano wpisywanie odwrotne
		
			FOR i := iEntranceArrayElements TO 1 BY -1 DO
				IF  NOT eExitState[i].bFormPresent THEN  		// Jeżeli w rejestrze wyjściowym jest wolne miejsce to wpisz rejestr wejściowy
					eExitState[i] := eEntranceState[1];	// Wpisz do rejestru dane np z [1] Buffor do [1,2,3,4,5,6] Package
					eEntranceState[1]:=eClearPackageState;	// Czyszczenie pierwszego rejestru wejściowego
					k:=i;											// Przepisywanie zmiennej pomocniczej
					FOR i := 1 TO iEntranceArrayElements DO   				
						IF i = iEntranceArrayElements THEN
							eEntranceState[i]:=eClearPackageState;		  // Zerowanie ostatniego bo zostało przesuniete wszystko o 1
						ELSE													  // Przepisanie 2 do 1, 3 do 2, 4 do 3, 5 do 4, 6 do 5, zeruj 6
							eEntranceState[i] := eEntranceState[i+1]; // 2 do 1, 3 do 2,
							eEntranceState[i+1]:=eClearPackageState;		  // zeruj 2, 
						END_IF
					END_FOR
					bTriggerDone := TRUE;
					EXIT;
					bError := TRUE;
					iError := 1;
				ELSE
					nFormCounter := nFormCounter + 1;
					bError := TRUE;
					iError := 2;
				END_IF
			END_FOR

		END_IF
		IF nFormCounter = iExitArrayElements THEN
		bKeepTryingMove:=NOT bNoKeepTryingMove;
		END_IF
	END_IF
ELSIF iEntranceArrayElements > iExitArrayElements AND bFirstCycle AND NOT bMoveOnlyToLastExitRegister THEN
	IF rtbTrigger.Q OR bKeepTryingMove OR bTriggerCounter THEN
		bTriggerCounter := FALSE; 
		bKeepTryingMove := FALSE;
		nFormCounter :=0;
		bBottlePresent := bCapPresent := FALSE; 
		IF NOT bInvertWriting THEN // Jezeli odwrotne wpisywanie
			FOR i := 1 TO iExitArrayElements DO
				IF  NOT eExitState[i].bFormPresent THEN  		// Jeżeli w rejestrze wyjściowym jest wolne miejsce to wpisz rejestr wejściowy
					eExitState[i] := eEntranceState[1];			// Wpisz do rejestru dane np z [1] Buffor do [1,2,3,4,5,6] Package
					eEntranceState[1]:=eClearPackageState;		// Czyszczenie pierwszego rejestru wejściowego
					k:=i;										// Przepisywanie zmiennej pomocniczej
					FOR i := 1 TO iEntranceArrayElements DO   				
						IF i = iEntranceArrayElements THEN
							eEntranceState[i]:=eClearPackageState;			// Zerowanie ostatniego bo zostało przesuniete wszystko o 1
						ELSE												// Przepisanie 2 do 1, 3 do 2, 4 do 3, 5 do 4, 6 do 5, zeruj 6
							IF NOT bMoveOnlyIfFormPresent THEN //ZMIANA LU192
								eEntranceState[i] := eEntranceState[i+1]; 		// 2 do 1, 3 do 2,
								eEntranceState[i+1]:=eClearPackageState;		// zeruj 2, 
							ELSE
								IF eEntranceState[i+1] .bFormPresent THEN
									eEntranceState[i] := eEntranceState[i+1]; 		// 2 do 1, 3 do 2,
									eEntranceState[i+1]:=eClearPackageState;		// zeruj 2, 	
								END_IF
							END_IF
						END_IF
					END_FOR
					bTriggerDone := TRUE;
					EXIT; 
					bError := TRUE;
					iError := 3;
				ELSE
					nFormCounter := nFormCounter + 1;
					bError := TRUE;
					iError := 4;
				END_IF
			END_FOR
		ELSE
			FOR i := iExitArrayElements TO 1 BY -1 DO
				IF  NOT eExitState[i].bFormPresent THEN  		// Jeżeli w rejestrze wyjściowym jest wolne miejsce to wpisz rejestr wejściowy
					eExitState[i] := eEntranceState[1];			// Wpisz do rejestru dane np z [1] Buffor do [1,2,3,4,5,6] Package
					eEntranceState[1]:=eClearPackageState;		// Czyszczenie pierwszego rejestru wejściowego
					k:=i;										// Przepisywanie zmiennej pomocniczej
					FOR i := 1 TO iEntranceArrayElements DO   				
						IF i = iEntranceArrayElements THEN
							eEntranceState[i]:=eClearPackageState;			// Zerowanie ostatniego bo zostało przesuniete wszystko o 1
						ELSE												// Przepisanie 2 do 1, 3 do 2, 4 do 3, 5 do 4, 6 do 5, zeruj 6
							eEntranceState[i] := eEntranceState[i+1]; 		// 2 do 1, 3 do 2,
							eEntranceState[i+1]:=eClearPackageState;		// zeruj 2, 
						END_IF
					END_FOR
					bTriggerDone := TRUE;
					EXIT;
					bError := TRUE;
					iError := 3;
				ELSE
					nFormCounter := nFormCounter + 1;
					bError := TRUE;
					iError := 4;
				END_IF
			END_FOR
		END_IF
	
		IF nFormCounter = iExitArrayElements THEN
			bKeepTryingMove:=NOT bNoKeepTryingMove;									
		END_IF																	
	END_IF
ELSIF iEntranceArrayElements < iExitArrayElements AND bFirstCycle AND NOT bMoveOnlyToLastExitRegister THEN
		IF rtbTrigger.Q OR bKeepTryingMove OR bTriggerCounter THEN
		bTriggerCounter := FALSE; 
		bKeepTryingMove := FALSE;
		nFormCounter := 0;
		(*Do testów - jeszcze raz nadpisz jakby czujniki były przestawione LU205*)	
		IF bCapPresent THEN		
			eEntranceState[1].bCapPutted := TRUE;
			eEntranceState[1].bCapOK := TRUE; eEntranceState[1].bBottlePresent:= TRUE;//Zmiana nowa
			eEntranceState[1].bFormPresent := TRUE;
		END_IF
		(*Koniec Do testów - jeszcze raz nadpisz jakby czujniki były przestawione*)

		bBottlePresent := bCapPresent  := FALSE; 
		IF NOT bInvertWriting AND NOT bRotateEntranceRegisterBefore THEN // Jezeli odwrotne wpisywanie
			FOR i := 1 TO iExitArrayElements DO
				IF  NOT eExitState[i].bFormPresent THEN  		// Jeżeli w rejestrze wyjściowym jest wolne miejsce to wpisz rejestr wejściowy
					eExitState[i] := eEntranceState[1];			// Wpisz do rejestru dane np z [1] Buffor do [1,2,3,4,5,6] Package
					eEntranceState[1]:=eClearPackageState;		// Czyszczenie pierwszego rejestru wejściowego
					k:=i;										// Przepisywanie zmiennej pomocniczej
					FOR i := 1 TO iEntranceArrayElements DO   				
						IF i = iEntranceArrayElements THEN
							eEntranceState[i]:=eClearPackageState;			// Zerowanie ostatniego bo zostało przesuniete wszystko o 1
						ELSE												// Przepisanie 2 do 1, 3 do 2, 4 do 3, 5 do 4, 6 do 5, zeruj 6
							eEntranceState[i] := eEntranceState[i+1]; 		// 2 do 1, 3 do 2,
							eEntranceState[i+1]:= eClearPackageState;		// zeruj 2, 
						END_IF
					END_FOR
					bTriggerDone := TRUE;
					EXIT;
					bError := TRUE;
					iError := 5;
				ELSE
					nFormCounter := nFormCounter + 1;
					bError := TRUE;
					iError := 6;
				END_IF
			END_FOR
		ELSIF bInvertWriting AND NOT bRotateEntranceRegisterBefore THEN
			FOR i := iExitArrayElements TO 1 BY -1 DO
				IF  NOT eExitState[i].bFormPresent THEN  		// Jeżeli w rejestrze wyjściowym jest wolne miejsce to wpisz rejestr wejściowy
					eExitState[i] := eEntranceState[1];			// Wpisz do rejestru dane np z [1] Buffor do [1,2,3,4,5,6] Package
					eEntranceState[1]:=eClearPackageState;		// Czyszczenie pierwszego rejestru wejściowego
					k:=i;										// Przepisywanie zmiennej pomocniczej
					FOR i := 1 TO iEntranceArrayElements DO   				
						IF i = iEntranceArrayElements THEN
							eEntranceState[i]:=eClearPackageState;			// Zerowanie ostatniego bo zostało przesuniete wszystko o 1
						ELSE												// Przepisanie 2 do 1, 3 do 2, 4 do 3, 5 do 4, 6 do 5, zeruj 6
							eEntranceState[i] := eEntranceState[i+1]; 		// 2 do 1, 3 do 2,
							eEntranceState[i+1]:= eClearPackageState;		// zeruj 2, 
						END_IF
					END_FOR
					bTriggerDone := TRUE;
					EXIT;
					bError := TRUE;
					iError := 5;
				ELSE
					nFormCounter := nFormCounter + 1;
					bError := TRUE;
					iError := 6;
				END_IF
			END_FOR
		ELSIF NOT bInvertWriting AND bRotateEntranceRegisterBefore THEN //Opcja najpierw przepisz a potem zabierz 
			FOR i := 1 TO iExitArrayElements DO
				IF  NOT eExitState[i].bFormPresent THEN  		// Jeżeli w rejestrze wyjściowym jest wolne miejsce to wpisz rejestr wejściowy
																// Przepisywanie zmiennej pomocniczej
					FOR j := 1 TO iEntranceArrayElements DO   				
						IF j = iEntranceArrayElements THEN
							eEntranceState[j]:=eClearPackageState;			// Zerowanie ostatniego bo zostało przesuniete wszystko o 1
						ELSE												// Przepisanie 2 do 1, 3 do 2, 4 do 3, 5 do 4, 6 do 5, zeruj 6
							eEntranceState[j] := eEntranceState[j+1]; 		// 2 do 1, 3 do 2,
							eEntranceState[j+1]:= eClearPackageState;		// zeruj 2, 
						END_IF
					END_FOR
					
					eExitState[i] := eEntranceState[1];			// Wpisz do rejestru dane np z [1] Buffor do [1,2,3,4,5,6] Package
					eEntranceState[1]:=eClearPackageState;		// Czyszczenie pierwszego rejestru wejściowego
					k:=i;
					
					bTriggerDone := TRUE;
					EXIT;
					bError := TRUE;
					iError := 5;
				ELSE
					nFormCounter := nFormCounter + 1;
					bError := TRUE;
					iError := 6;
				END_IF
			END_FOR
		END_IF
		IF nFormCounter = iExitArrayElements THEN
			bKeepTryingMove:=NOT bNoKeepTryingMove;
		END_IF
	END_IF
ELSIF bMoveOnlyToLastExitRegister THEN //Opcja wpisywania z rejestru wejsciowego na ostatni wyjsciowy bez przesuwania wyjsciowego 
		IF rtbTrigger.Q OR bKeepTryingMove OR bTriggerCounter THEN
		bTriggerCounter := FALSE; 
		bKeepTryingMove := FALSE;
		nFormCounter := 0;
		
		(*Do testów - jeszcze raz nadpisz jakby czujniki były przestawione LU205*)	
		IF bCapPresent THEN		
			eEntranceState[1].bCapPutted := TRUE;
			eEntranceState[1].bCapOK := TRUE; eEntranceState[1].bBottlePresent:= TRUE;//Zmiana nowa
			eEntranceState[1].bFormPresent := TRUE;
		END_IF
		(*Koniec Do testów - jeszcze raz nadpisz jakby czujniki były przestawione*)					
		bBottlePresent := bCapPresent := FALSE; 
		
				IF  NOT bWithCapControl AND NOT eExitState[iExitArrayElements].bFormPresent AND NOT bRotateEntranceRegisterBefore THEN  	// Jeżeli w rejestrze wyjściowym jest wolne miejsce to wpisz rejestr wejściowy
					eExitState[iExitArrayElements] := eEntranceState[1];	// Wpisz do rejestru dane np z [1] Buffor do [1,2,3,4,5,6] Package
					eEntranceState[1]:=eClearPackageState;		// Czyszczenie pierwszego rejestru wejściowego
					k:=i;										// Przepisywanie zmiennej pomocniczej
					FOR i := 1 TO iEntranceArrayElements DO   				
						IF i = iEntranceArrayElements THEN
							eEntranceState[i]:=eClearPackageState;			// Zerowanie ostatniego bo zostało przesuniete wszystko o 1
						ELSE												// Przepisanie 2 do 1, 3 do 2, 4 do 3, 5 do 4, 6 do 5, zeruj 6
							eEntranceState[i] := eEntranceState[i+1]; 		// 2 do 1, 3 do 2,
							eEntranceState[i+1]:= eClearPackageState;		// zeruj 2, 
						END_IF
					END_FOR
					bTriggerDone := TRUE;
					
					bError := TRUE;
					iError := 5;
				ELSIF bWithCapControl AND NOT bRotateEntranceRegisterBefore THEN //TUTAJ DODAŁEM
					eExitState[iExitArrayElements] := eEntranceState[1];	// Wpisz do rejestru dane np z [1] Buffor do [1,2,3,4,5,6] Package
					eEntranceState[1]:=eClearPackageState;		// Czyszczenie pierwszego rejestru wejściowego
					k:=i;										// Przepisywanie zmiennej pomocniczej
(*zmiana dp-1*)		FOR i := 1 TO iEntranceArrayElements DO   			
						IF i = iEntranceArrayElements THEN
							eEntranceState[i]:=eClearPackageState;			// Zerowanie ostatniego bo zostało przesuniete wszystko o 1
						ELSE												// Przepisanie 2 do 1, 3 do 2, 4 do 3, 5 do 4, 6 do 5, zeruj 6
							eEntranceState[i] := eEntranceState[i+1]; 		// 2 do 1, 3 do 2,
							eEntranceState[i+1]:= eClearPackageState;		// zeruj 2, 
						END_IF
					END_FOR
					bTriggerDone := TRUE;
					
				(*NEW*)	
				ELSIF NOT bInvertWriting AND bRotateEntranceRegisterBefore THEN //Opcja najpierw przepisz a potem zabierz 

							FOR j := 1 TO iEntranceArrayElements DO   				
								IF j = iEntranceArrayElements THEN
									eEntranceState[j]:=eClearPackageState;			// Zerowanie ostatniego bo zostało przesuniete wszystko o 1
								ELSE												// Przepisanie 2 do 1, 3 do 2, 4 do 3, 5 do 4, 6 do 5, zeruj 6
									eEntranceState[j] := eEntranceState[j+1]; 		// 2 do 1, 3 do 2,
									eEntranceState[j+1]:= eClearPackageState;		// zeruj 2, 
								END_IF
							END_FOR
							eExitState[iExitArrayElements] := eEntranceState[1];	// Wpisz do rejestru dane np z [1] Buffor do [1,2,3,4,5,6] Package
							eEntranceState[1]:=eClearPackageState;					// Czyszczenie pierwszego rejestru wejściowego
							bTriggerDone := TRUE;
							bError := TRUE;
							iError := 5;
		
				ELSE
					nFormCounter := nFormCounter + 1;
					bError := TRUE;
					iError := 6;
				END_IF				
				
			IF nFormCounter = 1 THEN
				bKeepTryingMove:=NOT bNoKeepTryingMove;
			END_IF
		END_IF
END_IF	


//CZYSZCZENIE REJESTRU WEJSCIOWEGO
IF rtbReset.Q THEN
	FOR r1 := 1 TO iEntranceArrayElements DO
		eEntranceState[r1] := eClearPackageState;
	END_FOR
	FOR r2 := 1 TO iExitArrayElements DO
		eExitState[r2] := eClearPackageState;
	END_FOR
	bKeepTryingMove :=FALSE;
	bTriggerDone := FALSE;
	bTriggerCounter := FALSE; 
	nFormCounter := 0;
	bBottlePresent := bCapPresent := FALSE; 
	bError := FALSE;
	iError := 0;
END_IF

END_FUNCTION_BLOCK

// ---- POUs/FB/FB_MoveRegister4.TcPOU
FUNCTION_BLOCK FB_MoveRegister4
VAR_INPUT
	bFirstCycle	:BOOL;						//Bit od pierwszego cyklu, żeby nie wykrywało zbocza opadającego
	bTrigger	:BOOL;						// BIt do wyzwalania przesuniecia o 4
	tTriggerFilterTimeOn	:TIME:=T#0MS;	// Czas filtrowania wejścia Trigger na załączenie
	tTriggerFilterTimeOFF	:TIME:=T#0MS;	// Czas filtorwania wejścia Trigger na wyłaczenie
	bInvertWriting: BOOL;					//Bit zapisu w odwrotenj kolejnosci
	bTriggerBottle	:BOOL;					// Zapisywanie czy butelka jest czy nie ( jeżeli jest włączona kontrola obecności)
	iEntrenceArrayElements	:UINT;			// Licznik ilości elementów w tablicy wejściowej
	iExitArrayElements	:UINT;				// Licznik ilosco elementów w tablicy wyjściowej
	bWithFormControlTrigerCounter	:BOOL;	// Jezeli na tr
	bMoveOnlyIfFormPresent	:BOOL;			//Przesuwanie tylko jeśli jest obecna formatka
	bMoveOnlyToLastExitRegister	:BOOL;		// PRzesuniecie tylko na ostatni rejstr wyjsciowy
	bMoveOnlyToLastRegister: BOOL;
	bNoKeepTryingMove: BOOL; 				//PRóbuj dakej przesunać jeżelei nie ma miejsca
	bReset	:BOOL;							// Czyszczenie tablicy
	eClearPackageState	:S_PackageState;	//Deklaracja czystego rejestru
	
	
	bRotateEntranceRegisterBefore: BOOL;	//Przesuwanie rejestrru wejściowego, a następnie go obrót
END_VAR
VAR_OUTPUT
	bError	:BOOL;	//Bład w sekwencji
	iError	:INT;	//Numer błędu 
	bTriggerDone :BOOL;		//Przesunięcie wykonane
	bTriggerFilteredOUT:BOOL;	//Sygnał przefiltorwanego bitu aktywacji przesuniecia 
END_VAR
VAR_IN_OUT
	bTriggerCounter	:BOOL;   //Triger do kasowania
	eEntranceState :ARRAY[1..17] OF S_PackageState;		//Tablica wejściowa danych
	eExitState	:ARRAY[1..17] OF S_PackageState;		//Tablica wyjściowa danych
	bKeepTryingMove	:BOOL;	//Próbuj zapisać formatki dalej, aż do zwolnienia miejsca
END_VAR
VAR
	tofTriggerFilterTimeOff: TOF;	//Czasówka do filtrowania wyzwolenia przesuniecia
	tonTriggerFilterTimeOn: TON;	// Czas do filtrowania wyzwolenia przesuniecia
	bTriggerFiltered: BOOL;		//Bit informujacy o przefiltrowaniu wejscai
	bWithBottleControl: BOOL;	// Bit od kontroli butleki
	rtbTrigger: R_TRIG;		//Bit zbocza narastającego przesuniecia formatki
	rtbTriggerBottle: R_TRIG;	// Bit zbocza narastającego butelki
	rtbReset: R_TRIG;
	bWithCapControl: BOOL;		//Bit kontroli obecnosci nasadki
	i: UINT;		//Licznik pętli
	nFormCounter: UINT; //Licznik formatek
	j: UINT;			//Zmienna pomocncza
	r1: UINT;			//Zmienna pomocnicza
	r2: UINT;			//Zmienna pomocnicza

	TimerResetErrors: TON;
	k: UINT;
	bNotEmptyPlace: BOOL;
END_VAR

//Filtrowanie sygnału wejściowego
tofTriggerFilterTimeOff	(IN:=bTrigger, PT:=tTriggerFilterTimeOff);
tonTriggerFilterTimeOn	(IN:=tofTriggerFilterTimeOff.Q, PT:=tTriggerFilterTimeOn);
bTriggerFiltered 		:= tonTriggerFilterTimeOn.Q;
bTriggerFilteredOUT		:= bTriggerFiltered ;

//TRIGI I TIMERY
IF bWithBottleControl THEN
	rtbTrigger 	(CLK := NOT bTriggerFiltered, Q=>);
	rtbTriggerBottle 	(CLK := NOT bTriggerBottle, Q=>);
ELSIF bWithCapControl THEN
	rtbTrigger 	(CLK := NOT bTriggerFiltered, Q=>);
ELSE
	rtbTrigger 	(CLK := bTriggerFiltered, Q=>);
	rtbTriggerBottle 	(CLK := bTriggerBottle, Q=>);
END_IF

rtbReset 	(CLK := bReset, Q=>);
TimerResetErrors (IN:= bError, PT:=T#1000MS, Q=>);

//RESETOWANIE BLEDU
IF TimerResetErrors.Q THEN
	bError := FALSE;
END_IF

bTriggerDone := FALSE;

// PRzesuniecie rejestrów 

IF iEntrenceArrayElements = iExitArrayElements AND  bFirstCycle THEN
	IF rtbTrigger.Q OR bKeepTryingMove THEN
		bTriggerCounter	:=FALSE;
		bKeepTryingMove	:=FALSE;
		bNotEmptyPlace:=FALSE;
		nFormCounter:=0;
		
		eExitState[1]:= eEntranceState[1];
		eExitState[2]:= eEntranceState[2];
		eExitState[3]:= eEntranceState[3];
		eExitState[4]:= eEntranceState[4];
		
		eEntranceState[1]:=eClearPackageState;
		eEntranceState[2]:=eClearPackageState;
		eEntranceState[3]:=eClearPackageState;
		eEntranceState[4]:=eClearPackageState;
		
		END_IF
	END_IF




//CZYSZCZENIE REJESTRU WEJSCIOWEGO
IF rtbReset.Q THEN
	FOR r1 := 1 TO iEntrenceArrayElements DO
		eEntranceState[r1] := eClearPackageState;
	END_FOR
	FOR r2 := 1 TO iExitArrayElements DO
		eExitState[r2] := eClearPackageState;
	END_FOR
	bKeepTryingMove :=FALSE;
	bTriggerDone := FALSE;
	bTriggerCounter := FALSE; 
	nFormCounter := 0;
	//bBottlePresent := bCapPresent := FALSE; 
	bError := FALSE;
	iError := 0;
END_IF

END_FUNCTION_BLOCK

// ---- POUs/FB/FB_MoveRegisterSortAndMove.TcPOU
(*
Nazwa:			FB_MoveRegister
Opis:			Blok przesuniecia rejestru formatek
Wersja:			v0.3 		
Data:			2018-11-16
Autor:			DP
Urzadzenia:		 
Konfiguracja:	
Info:
- Są dwa rejestry, wejściowy i wyjsciowy (struktury)
- Jezeli rejestr ma np. 6 elementów to za kazdym razem po wykryciu trigera program będzie
	1 wejściowy przesuwał na 1 wolny (nie ma formatki) wyjściowy
	kasował 1 rejestr wejściowy
	przesuwal rejetr wejsciowy 2 na 1(przeniesiony i skasowany), 3 na 2, 4 na 3, 5 na 4, 6 na 5 i kasowal 6wejsciowy
	tym sposobem po 6 trigerach caly rejestr wejsciowy powinien być na wyjsciowym
	np po 3 trigerach na wyjsciowym powinny byc zajete 1 do 3 i na wejsciowym 1 do 3
Błędy:
1 - nie wyszło z pętli for
2 - formatka już jest w rejestrze
Uwagi:
- 
Zmiany:
2018-09-18 Dodano sprawdzanie nasadek
2018-06-14 DP Pierwsza wersja
*)

FUNCTION_BLOCK FB_MoveRegisterSortAndMove
VAR_INPUT
	bFirstCycle:BOOL;					//Pierwszy cykl, zeby na początku nie wykrywało zbocza opadającego
	bTrigger :BOOL;						// Przesuniecie tablicy o jeden
	tTriggerFilterTimeOn:TIME:=T#0MS;	// Czas filtrowania wejścia Trigger na załączenie
	tTriggerFilterTimeOff:TIME:=T#0MS;	// Czas filtrowania wejścia Trigger na wyłączenie
	bTriggerBottle :BOOL;				// Zapisywanie czy jest butelka czy nie (jezeli kontrola wlączona)
	bWithBottleControl: BOOL;			// Włączona opcja kontroli butelek
	bWithCapControl:BOOL;				// Wlaczona kontrola nasadek
	bWithFormControlTrigerCounter:BOOL;	// Jezeku na trigercontrol nie ma formatki do przesunięcia to stwórz nową
	bMoveOnlyIfFormPresent:BOOL;		// Przepisuj tylko jak jest formatka
	bRotateEntranceRegisterBefore:BOOL;	// Najpierw przesuń rejestr wejściowy a następnie z niego zabierz
	bNoKeepTryingMove:BOOL;				// Dalej przepisuj jezeli nie ma miejsca
	bTriggerCap: BOOL;					// Truger wykrycia nasadki
	bReset :BOOL;						// Czyszczenie tablic
	iEntranceArrayElements :UINT; 		// Wartość koncowa tablicy
	iExitArrayElements :UINT; 			// Wartość koncowa tablicy
	bInvertWriting :BOOL;				// Wpisywanie odwrotne zamist z 1entrance na 1exit to 1entrance na 6exit	
	eClearPackageState :S_PackageState; // Czysty rejestr
END_VAR
VAR_IN_OUT
	bTriggerCounter :BOOL;		// Triger ktory jest kasowany
	eEntranceState :ARRAY [1..17] OF S_PackageState;	
	eExitState :ARRAY [1..17] OF S_PackageState;
	bKeepTryingMove :BOOL;		// Probuj dalej zapisać formatki aż się któraś zwolni
END_VAR

VAR_OUTPUT	
	bError :BOOL; 				// Błąd
	iError: UINT;				// Nr Błędu
	bTriggerDone :BOOL; 		// Wykonano przesunięcie
	bTriggerFilteredOUT:BOOL;	//Wyjscie przefiltrowanego sygnalu wejsciowego
END_VAR

VAR
	i:UINT;						// Zmienna w tablicy
	k:UINT;						// Pomocnicza zmienna do zapisywnia czy jest butelka
	rtbTrigger :R_TRIG;			// Reaguje na zbocze
	rtbTriggerBottle :R_TRIG;	// Reaguje na zbocze
	rtbReset :R_TRIG;			// Reaguje na zbocze
	TimerResetErrors :TON;		// Reset Błedu
	nFormCounter :UINT;					//Licznik formatek
	r1,r2:UINT;
	bBottlePresent: BOOL;				//Zmienna pomocnicza ze wykryto butelkę
	bCapPresent: BOOL;					//Zmienna pomocnicza ze wykryto butelkę
	j: UINT;
	tonTriggerFilterTimeOn: TON;
	bTriggerFiltered: BOOL;
	tofTriggerFilterTimeOff: TOF;
END_VAR

//Filtrowanie sygnału wejściowego
tofTriggerFilterTimeOff	(IN:=bTrigger, PT:=tTriggerFilterTimeOff);
tonTriggerFilterTimeOn	(IN:=tofTriggerFilterTimeOff.Q, PT:=tTriggerFilterTimeOn);
bTriggerFiltered 		:= tonTriggerFilterTimeOn.Q;
bTriggerFilteredOUT		:= bTriggerFiltered ;

//TRIGI I TIMERY
IF bWithBottleControl THEN
	rtbTrigger 	(CLK := NOT bTriggerFiltered, Q=>);
	rtbTriggerBottle 	(CLK := NOT bTriggerBottle, Q=>);
ELSIF bWithCapControl THEN
	rtbTrigger 	(CLK := NOT bTriggerFiltered, Q=>);
ELSE
	rtbTrigger 	(CLK := bTriggerFiltered, Q=>);
	rtbTriggerBottle 	(CLK := bTriggerBottle, Q=>);
END_IF

rtbReset 	(CLK := bReset, Q=>);
TimerResetErrors (IN:= bError, PT:=T#1000MS, Q=>);

//RESETOWANIE BLEDU
IF TimerResetErrors.Q THEN
	bError := FALSE;
END_IF

//KASOWANIE ZMIENNYCH
bTriggerDone := FALSE;

//JEZELI WLACZONO KONTROLE BUTELEK TO NADPISUJ REJESTR CZY JEST BUTELKA
IF bWithBottleControl AND bTrigger AND bTriggerBottle AND NOT bKeepTryingMove THEN //Jezeli od wykrycia formatki liczy TIMER i wykryło butelke to wpisz do rejestru że jest butelka
	eEntranceState[1].bBottlePresent := TRUE;
	eEntranceState[1].bFormPresent := TRUE;
	bBottlePresent := TRUE; // Wpisuje że jest butelka jezeli wystąpi sygnał podczas trwania czujnika formatki
ELSIF bWithBottleControl AND rtbTrigger.Q AND NOT bBottlePresent AND  NOT bKeepTryingMove AND bFirstCycle THEN
	eEntranceState[1].bBottlePresent := FALSE;
	eEntranceState[1].bFormPresent := TRUE; // jeżeli zanik czujnik formatki i nie było formatki to wpisz ze nie było butelki
END_IF
//JEZELI WLACZONO KONTROLE NASADEk TO NADPISUJ REJESTR CZY JEST BUTELKA 
(*IF bWithCapControl AND bTrigger AND bTriggerCap AND NOT bKeepTryingMove THEN //Jezeli od wykrycia formatki liczy TIMER i wykryło butelke to wpisz do rejestru że jest butelka
	eEntranceState[1].bCapPutted := TRUE;
	eEntranceState[1].bCapOK := TRUE; eEntranceState[1].bBottlePresent:= TRUE;//Zmiana nowa
	eEntranceState[1].bFormPresent := TRUE;
	bCapPresent := TRUE; // Wpisuje że jest butelka jezeli wystąpi sygnał podczas trwania czujnika formatki*)
	//ZMIANA LU 192
IF bWithCapControl AND bTriggerCap AND NOT bKeepTryingMove THEN //Jezeli od wykrycia formatki liczy TIMER i wykryło butelke to wpisz do rejestru że jest butelka
	eEntranceState[1].bCapPutted := TRUE;
	eEntranceState[1].bCapOK := TRUE; eEntranceState[1].bBottlePresent:= TRUE;//Zmiana nowa
	eEntranceState[1].bFormPresent := TRUE;
	bCapPresent := TRUE; // Wpisuje że jest butelka jezeli wystąpi sygnał podczas trwania czujnika formatki	
ELSIF bWithCapControl AND rtbTrigger.Q AND NOT bCapPresent AND  NOT bKeepTryingMove AND bFirstCycle THEN
	eEntranceState[1].bCapPutted := TRUE;
	eEntranceState[1].bCapOK:= FALSE;
	eEntranceState[1].bFormPresent := TRUE; // jeżeli zanik czujnik formatki i nie było formatki to wpisz ze nie było butelki
END_IF
//JEZELI WLACZONO SPRAWDZANIE FORMATEK Z TRIGERCOUNTER TO
IF bWithFormControlTrigerCounter  AND bTriggerCounter AND NOT bKeepTryingMove AND bFirstCycle THEN
	eEntranceState[1].bFormPresent := TRUE;
END_IF



//PRZESUNIECIE
IF iEntranceArrayElements <= iExitArrayElements AND bFirstCycle  THEN
		IF rtbTrigger.Q OR bKeepTryingMove OR bTriggerCounter THEN
		bTriggerCounter := FALSE; 
		bKeepTryingMove := FALSE;
		nFormCounter := 0;
		bBottlePresent := bCapPresent  := FALSE; 
		FOR i:= 1 TO iExitArrayElements-1 DO // SORTOWANIE
			IF NOT eExitState[i].bFormPresent THEN 
				eExitState[i] := eExitState[i+1];
				eExitState[i+1] := eClearPackageState;
			END_IF
		END_FOR

		FOR i := 1 TO iExitArrayElements DO
			IF  NOT eExitState[i].bFormPresent THEN  		// Jeżeli w rejestrze wyjściowym jest wolne miejsce to wpisz rejestr wejściowy
				eExitState[i] := eEntranceState[1];			// Wpisz do rejestru dane np z [1] Buffor do [1,2,3,4,5,6] Package
				eEntranceState[1]:=eClearPackageState;		// Czyszczenie pierwszego rejestru wejściowego
				k:=i;										// Przepisywanie zmiennej pomocniczej
				FOR i := 1 TO iEntranceArrayElements DO   				
					IF i = iEntranceArrayElements THEN
						eEntranceState[i]:=eClearPackageState;			// Zerowanie ostatniego bo zostało przesuniete wszystko o 1
					ELSE												// Przepisanie 2 do 1, 3 do 2, 4 do 3, 5 do 4, 6 do 5, zeruj 6
						eEntranceState[i] := eEntranceState[i+1]; 		// 2 do 1, 3 do 2,
						eEntranceState[i+1]:= eClearPackageState;		// zeruj 2, 
					END_IF
				END_FOR
				bTriggerDone := TRUE;
				EXIT;
				bError := TRUE;
				iError := 5;
			ELSE
				nFormCounter := nFormCounter + 1;
				bError := TRUE;
				iError := 6;
			END_IF
		END_FOR

		IF nFormCounter = iExitArrayElements THEN
			bKeepTryingMove:=NOT bNoKeepTryingMove;
		END_IF
	END_IF
END_IF


//CZYSZCZENIE REJESTRU WEJSCIOWEGO
IF rtbReset.Q THEN
	FOR r1 := 1 TO iEntranceArrayElements DO
		eEntranceState[r1] := eClearPackageState;
	END_FOR
	FOR r2 := 1 TO iExitArrayElements DO
		eExitState[r2] := eClearPackageState;
	END_FOR
	bKeepTryingMove :=FALSE;
	bTriggerDone := FALSE;
	bTriggerCounter := FALSE; 
	nFormCounter := 0;
	bBottlePresent := bCapPresent := FALSE; 
	bError := FALSE;
	iError := 0;
END_IF

END_FUNCTION_BLOCK

// ---- POUs/FB/FB_MoveRegisterCapControl.TcPOU
(*
Nazwa:			FB_MoveRegister
Opis:			Blok przesuniecia rejestru formatek
Wersja:			v0.3 		
Data:			2018-11-16
Autor:			DP
Urzadzenia:		 
Konfiguracja:	
Info:
- Są dwa rejestry, wejściowy i wyjsciowy (struktury)
- Jezeli rejestr ma np. 6 elementów to za kazdym razem po wykryciu trigera program będzie
	1 wejściowy przesuwał na 1 wolny (nie ma formatki) wyjściowy
	kasował 1 rejestr wejściowy
	przesuwal rejetr wejsciowy 2 na 1(przeniesiony i skasowany), 3 na 2, 4 na 3, 5 na 4, 6 na 5 i kasowal 6wejsciowy
	tym sposobem po 6 trigerach caly rejestr wejsciowy powinien być na wyjsciowym
	np po 3 trigerach na wyjsciowym powinny byc zajete 1 do 3 i na wejsciowym 1 do 3
Błędy:
1 - nie wyszło z pętli for
2 - formatka już jest w rejestrze
Uwagi:
- 
Zmiany:
2018-09-18 Dodano sprawdzanie nasadek
2018-06-14 DP Pierwsza wersja
*)

FUNCTION_BLOCK FB_MoveRegisterCapControl
VAR_INPUT
	bFirstCycle:BOOL;					//Pierwszy cykl, zeby na początku nie wykrywało zbocza opadającego
	bTrigger :BOOL;						// Przesuniecie tablicy o jeden
	tTriggerFilterTimeOn:TIME:=T#0MS;	// Czas filtrowania wejścia Trigger na załączenie
	tTriggerFilterTimeOff:TIME:=T#0MS;	// Czas filtrowania wejścia Trigger na wyłączenie
	bTriggerBottle :BOOL;				// Zapisywanie czy jest butelka czy nie (jezeli kontrola wlączona)
	bWithBottleControl: BOOL;			// Włączona opcja kontroli butelek
	bWithCapControl:BOOL;				// Wlaczona kontrola nasadek
	bWithFormControlTrigerCounter:BOOL;	// Jezeku na trigercontrol nie ma formatki do przesunięcia to stwórz nową
	bNoKeepTryingMove:BOOL;				// Dalej przepisuj jezeli nie ma miejsca
	bTriggerCap: BOOL;					// Truger wykrycia nasadki
	bReset :BOOL;						// Czyszczenie tablic
	iEntranceArrayElements :UINT; 		// Wartość koncowa tablicy
	iExitArrayElements :UINT; 			// Wartość koncowa tablicy
	eClearPackageState :S_PackageState; // Czysty rejestr
END_VAR
VAR_IN_OUT
	eEntranceState :ARRAY [1..17] OF S_PackageState;	
	eExitState :ARRAY [1..17] OF S_PackageState;
	iBottleWithoutCap: INT;
	bKeepTryingMove :BOOL;		// Probuj dalej zapisać formatki aż się któraś zwolni
	bRFIDReaded :BOOL;
END_VAR

VAR_OUTPUT	
	bError :BOOL; 				// Błąd
	iError: UINT;				// Nr Błędu
	bTriggerDone :BOOL; 		// Wykonano przesunięcie

	bTriggerFilteredOUT:BOOL;	//Wyjscie przefiltrowanego sygnalu wejsciowego
END_VAR

VAR
	i:UINT;						// Zmienna w tablicy
	k:UINT;						// Pomocnicza zmienna do zapisywnia czy jest butelka
	rtbTrigger :R_TRIG;			// Reaguje na zbocze
	rtbTriggerBottle :R_TRIG;	// Reaguje na zbocze
	rtbReset :R_TRIG;			// Reaguje na zbocze
	TimerResetErrors :TON;		// Reset Błedu
	nFormCounter :UINT;					//Licznik formatek
	r1,r2:UINT;
	bBottlePresent: BOOL;				//Zmienna pomocnicza ze wykryto butelkę
	bCapPresent: BOOL;					//Zmienna pomocnicza ze wykryto butelkę
	j: UINT;
	tonTriggerFilterTimeOn: TON;
	bTriggerFiltered: BOOL;
	tofTriggerFilterTimeOff: TOF;
	fbTriggerFiltered: FB_InputFIlter;
	ftfbTriggerFiltered: F_TRIG;
	tpTrigger: TP;
END_VAR

//Filtrowanie sygnału wejściowego
fbTriggerFiltered		(bIN:= 	bTrigger AND bRFIDReaded,		tFilterTimeOn:=tTriggerFilterTimeOn,	tFilterTimeOff:=tTriggerFilterTimeOff);
tpTrigger				(IN:=bTrigger, 		PT:=T#10MS);
bTriggerFilteredOUT		:= fbTriggerFiltered.bOUT ;

//TRIGI I TIMERY
ftfbTriggerFiltered		(CLK:=	fbTriggerFiltered.bOUT, 	Q=>);

rtbReset 				(CLK := bReset, Q=>);
TimerResetErrors 		(IN:= bError, PT:=T#1000MS, Q=>);

//RESETOWANIE BLEDU
IF TimerResetErrors.Q THEN
	bError := FALSE;
END_IF

//KASOWANIE ZMIENNYCH
bTriggerDone := FALSE;

//JEZELI WLACZONO KONTROLE NASADEk TO NADPISUJ REJESTR CZY JEST BUTELKA 
IF bWithCapControl AND bTriggerCap AND NOT bKeepTryingMove THEN //Jezeli od wykrycia formatki liczy TIMER i wykryło butelke to wpisz do rejestru że jest butelka
	eEntranceState[1].bCapPutted := TRUE;
	eEntranceState[1].bCapOK := TRUE; eEntranceState[1].bBottlePresent:= TRUE;//Zmiana nowa
	bCapPresent := TRUE; // Wpisuje że jest butelka jezeli wystąpi sygnał podczas trwania czujnika formatki	
ELSIF bWithCapControl AND ftfbTriggerFiltered.Q AND NOT bCapPresent AND  NOT bKeepTryingMove AND bFirstCycle THEN
	eEntranceState[1].bCapPutted := TRUE;
	eEntranceState[1].bCapOK:= FALSE;
END_IF
//JEZELI WLACZONO SPRAWDZANIE FORMATEK Z TRIGERCOUNTER TO
IF  tpTrigger.Q AND NOT bKeepTryingMove AND bFirstCycle THEN //Zmiena UBL50, tworz tez nowa jak Trigger
	eEntranceState[1].bFormPresent := TRUE;
END_IF

//PRZESUNIECIE
IF iEntranceArrayElements < iExitArrayElements AND bFirstCycle THEN
	IF ftfbTriggerFiltered.Q OR bKeepTryingMove THEN
		bRFIDReaded		:= FALSE;
		bKeepTryingMove := FALSE;
		nFormCounter := 0;
		(*Do testów - jeszcze raz nadpisz jakby czujniki były przestawione LU205*)	
		IF bCapPresent THEN		
			eEntranceState[1].bCapPutted := TRUE;
			eEntranceState[1].bCapOK := TRUE; eEntranceState[1].bBottlePresent:= TRUE;//Zmiana nowa
			eEntranceState[1].bFormPresent := TRUE;
		END_IF
		(*Koniec Do testów - jeszcze raz nadpisz jakby czujniki były przestawione*)

		bBottlePresent := bCapPresent  := FALSE; 
		FOR i:= 1 TO iExitArrayElements-1 DO // SORTOWANIE
			IF NOT eExitState[i].bFormPresent THEN 
				eExitState[i] := eExitState[i+1];
				eExitState[i+1] := eClearPackageState;
			END_IF
		END_FOR
		FOR i := 1 TO iExitArrayElements DO
			IF  NOT eExitState[i].bFormPresent THEN  		// Jeżeli w rejestrze wyjściowym jest wolne miejsce to wpisz rejestr wejściowy
				eExitState[i] 		:= 	eEntranceState[1];			// Wpisz do rejestru dane np z [1] Buffor do [1,2,3,4,5,6] Package
				eEntranceState[1]	:=	eClearPackageState;		// Czyszczenie pierwszego rejestru wejściowego
				k:=i;										// Przepisywanie zmiennej pomocniczej
				bTriggerDone := TRUE;
				IF eExitState[i].bBottlePresent AND NOT eExitState[i].bCapOK THEN
					iBottleWithoutCap	:=	iBottleWithoutCap	+1;
				END_IF
				IF eExitState[i].bBottlePresent AND eExitState[i].bCapOK THEN
					iBottleWithoutCap	:=	0;	
				END_IF	
				IF NOT eExitState[i].bBottlePresent THEN
					iBottleWithoutCap	:=	0;	
				END_IF				
				EXIT;
				bError := TRUE;
				iError := 5;
			ELSE
				nFormCounter := nFormCounter + 1;
				bError := TRUE;
				iError := 6;
			END_IF
		END_FOR
		IF nFormCounter = iExitArrayElements THEN
			bKeepTryingMove:=NOT bNoKeepTryingMove;
		END_IF
	END_IF
END_IF

//CZYSZCZENIE REJESTRU WEJSCIOWEGO
IF rtbReset.Q THEN
	FOR r1 := 1 TO iEntranceArrayElements DO
		eEntranceState[r1] := eClearPackageState;
	END_FOR
	FOR r2 := 1 TO iExitArrayElements DO
		eExitState[r2] := eClearPackageState;
	END_FOR
	bKeepTryingMove :=FALSE;
	bTriggerDone := FALSE;
	nFormCounter := 0;
	bBottlePresent := bCapPresent := FALSE; 
	bError := FALSE;
	iError := 0;
END_IF

END_FUNCTION_BLOCK

// ---- POUs/FB/FB_InputFilter.TcPOU
(*
Nazwa:			FB_InputFilter
Opis: 			Filtrowanie czujnikow
Wersja:			v1.0
Data:			2023-09-20
Autor:			DP
Urzadzenia:		
Konfiguracja:	
Info:
- blok filtrujacy wejście cyfrowe
*)

FUNCTION_BLOCK FB_InputFilter
VAR_INPUT
	bIN:BOOL;				//Wejście cyfrowe
	tFilterTimeOn:TIME;		//Czas filtrowania
	tFilterTimeOff:TIME;	//Czas filtrowania
END_VAR
VAR_OUTPUT
	bOUT:BOOL;
END_VAR
VAR
	tonIN: TON;
	tonOFF: TOF;
END_VAR


(* w1
tonOFF(IN:=bIN, PT:=tFilterTimeOff);
tonIN(IN:=tonOFF.Q, PT:=tFilterTimeOn);
bOUT:=tonIN.Q;
*)

(* w2 *)
tonIN	(IN:=bIN, 		PT:=tFilterTimeOn);
tonOFF	(IN:=NOT bIN, 	PT:=tFilterTimeOff);
IF tonIN.Q THEN
	bOUT := 	TRUE;
ELSIF tonOFF.Q THEN
	bOUT := 	FALSE;
END_IF

END_FUNCTION_BLOCK

// ---- POUs/FB/FB_MoveRegisterSortAndMoveLF.TcPOU
(*
Nazwa:			FB_MoveRegister
Opis:			Blok przesuniecia rejestru formatek
Wersja:			v0.3 		
Data:			2018-11-16
Autor:			DP
Urzadzenia:		 
Konfiguracja:	
Info:
- Są dwa rejestry, wejściowy i wyjsciowy (struktury)
- Jezeli rejestr ma np. 6 elementów to za kazdym razem po wykryciu trigera program będzie
	1 wejściowy przesuwał na 1 wolny (nie ma formatki) wyjściowy
	kasował 1 rejestr wejściowy
	przesuwal rejetr wejsciowy 2 na 1(przeniesiony i skasowany), 3 na 2, 4 na 3, 5 na 4, 6 na 5 i kasowal 6wejsciowy
	tym sposobem po 6 trigerach caly rejestr wejsciowy powinien być na wyjsciowym
	np po 3 trigerach na wyjsciowym powinny byc zajete 1 do 3 i na wejsciowym 1 do 3
Błędy:
1 - nie wyszło z pętli for
2 - formatka już jest w rejestrze
Uwagi:
- 
Zmiany:
2018-09-18 Dodano sprawdzanie nasadek
2018-06-14 DP Pierwsza wersja
*)

FUNCTION_BLOCK FB_MoveRegisterSortAndMoveLF
VAR_INPUT
	bFirstCycle:BOOL;					//Pierwszy cykl, zeby na początku nie wykrywało zbocza opadającego
	bTrigger :BOOL;						// Przesuniecie tablicy o jeden
	tTriggerFilterTimeOn:TIME:=T#0MS;	// Czas filtrowania wejścia Trigger na załączenie
	tTriggerFilterTimeOff:TIME:=T#0MS;	// Czas filtrowania wejścia Trigger na wyłączenie
	bTriggerBottle :BOOL;				// Zapisywanie czy jest butelka czy nie (jezeli kontrola wlączona)
	bWithBottleControl: BOOL;			// Włączona opcja kontroli butelek
	bWithCapControl:BOOL;				// Wlaczona kontrola nasadek
	bWithFormControlTrigerCounter:BOOL;	// Jezeku na trigercontrol nie ma formatki do przesunięcia to stwórz nową
	bMoveOnlyIfFormPresent:BOOL;		// Przepisuj tylko jak jest formatka
	bRotateEntranceRegisterBefore:BOOL;	// Najpierw przesuń rejestr wejściowy a następnie z niego zabierz
	bNoKeepTryingMove:BOOL;				// Dalej przepisuj jezeli nie ma miejsca
	bTriggerCap: BOOL;					// Truger wykrycia nasadki
	bReset :BOOL;						// Czyszczenie tablic
	iEntranceArrayElements :UINT; 		// Wartość koncowa tablicy
	iExitArrayElements :UINT; 			// Wartość koncowa tablicy
	bInvertWriting :BOOL;				// Wpisywanie odwrotne zamist z 1entrance na 1exit to 1entrance na 6exit	
	eClearPackageState :S_PackageState; // Czysty rejestr
END_VAR
VAR_IN_OUT
	bTriggerCounter :BOOL;		// Triger ktory jest kasowany
	eEntranceState :ARRAY [1..17] OF S_PackageState;	
	eExitState :ARRAY [1..17] OF S_PackageState;
	bKeepTryingMove :BOOL;		// Probuj dalej zapisać formatki aż się któraś zwolni
END_VAR

VAR_OUTPUT	
	bError :BOOL; 				// Błąd
	iError: UINT;				// Nr Błędu
	bTriggerDone :BOOL; 		// Wykonano przesunięcie
	bTriggerFilteredOUT:BOOL;	//Wyjscie przefiltrowanego sygnalu wejsciowego
END_VAR

VAR
	i:UINT;						// Zmienna w tablicy
	k:UINT;						// Pomocnicza zmienna do zapisywnia czy jest butelka
	rtbTrigger :R_TRIG;			// Reaguje na zbocze
	rtbTriggerBottle :R_TRIG;	// Reaguje na zbocze
	rtbReset :R_TRIG;			// Reaguje na zbocze
	TimerResetErrors :TON;		// Reset Błedu
	nFormCounter :UINT;					//Licznik formatek
	r1,r2:UINT;
	bBottlePresent: BOOL;				//Zmienna pomocnicza ze wykryto butelkę
	bCapPresent: BOOL;					//Zmienna pomocnicza ze wykryto butelkę
	j: UINT;
	tonTriggerFilterTimeOn: TON;
	bTriggerFiltered: BOOL;
	tofTriggerFilterTimeOff: TOF;
	iLFTest2: INT;
END_VAR

//Filtrowanie sygnału wejściowego
tofTriggerFilterTimeOff	(IN:=bTrigger, PT:=tTriggerFilterTimeOff);
tonTriggerFilterTimeOn	(IN:=tofTriggerFilterTimeOff.Q, PT:=tTriggerFilterTimeOn);
bTriggerFiltered 		:= tonTriggerFilterTimeOn.Q;
bTriggerFilteredOUT		:= bTriggerFiltered ;

//TRIGI I TIMERY
IF bWithBottleControl THEN
	rtbTrigger 	(CLK := NOT bTriggerFiltered, Q=>);
	rtbTriggerBottle 	(CLK := NOT bTriggerBottle, Q=>);
ELSIF bWithCapControl THEN
	rtbTrigger 	(CLK := NOT bTriggerFiltered, Q=>);
ELSE
	rtbTrigger 	(CLK := bTriggerFiltered, Q=>);
	rtbTriggerBottle 	(CLK := bTriggerBottle, Q=>);
END_IF

rtbReset 	(CLK := bReset, Q=>);
TimerResetErrors (IN:= bError, PT:=T#1000MS, Q=>);

//RESETOWANIE BLEDU
IF TimerResetErrors.Q THEN
	bError := FALSE;
END_IF

//KASOWANIE ZMIENNYCH
bTriggerDone := FALSE;

//JEZELI WLACZONO KONTROLE BUTELEK TO NADPISUJ REJESTR CZY JEST BUTELKA
IF bWithBottleControl AND bTrigger AND bTriggerBottle AND NOT bKeepTryingMove THEN //Jezeli od wykrycia formatki liczy TIMER i wykryło butelke to wpisz do rejestru że jest butelka
	eEntranceState[1].bBottlePresent := TRUE;
	eEntranceState[1].bFormPresent := TRUE;
	bBottlePresent := TRUE; // Wpisuje że jest butelka jezeli wystąpi sygnał podczas trwania czujnika formatki
ELSIF bWithBottleControl AND rtbTrigger.Q AND NOT bBottlePresent AND  NOT bKeepTryingMove AND bFirstCycle THEN
	eEntranceState[1].bBottlePresent := FALSE;
	eEntranceState[1].bFormPresent := TRUE; // jeżeli zanik czujnik formatki i nie było formatki to wpisz ze nie było butelki
END_IF
//JEZELI WLACZONO KONTROLE NASADEk TO NADPISUJ REJESTR CZY JEST BUTELKA 
(*IF bWithCapControl AND bTrigger AND bTriggerCap AND NOT bKeepTryingMove THEN //Jezeli od wykrycia formatki liczy TIMER i wykryło butelke to wpisz do rejestru że jest butelka
	eEntranceState[1].bCapPutted := TRUE;
	eEntranceState[1].bCapOK := TRUE; eEntranceState[1].bBottlePresent:= TRUE;//Zmiana nowa
	eEntranceState[1].bFormPresent := TRUE;
	bCapPresent := TRUE; // Wpisuje że jest butelka jezeli wystąpi sygnał podczas trwania czujnika formatki*)
	//ZMIANA LU 192
IF bWithCapControl AND bTriggerCap AND NOT bKeepTryingMove THEN //Jezeli od wykrycia formatki liczy TIMER i wykryło butelke to wpisz do rejestru że jest butelka
	eEntranceState[1].bCapPutted := TRUE;
	eEntranceState[1].bCapOK := TRUE; eEntranceState[1].bBottlePresent:= TRUE;//Zmiana nowa
	eEntranceState[1].bFormPresent := TRUE;
	bCapPresent := TRUE; // Wpisuje że jest butelka jezeli wystąpi sygnał podczas trwania czujnika formatki	
ELSIF bWithCapControl AND rtbTrigger.Q AND NOT bCapPresent AND  NOT bKeepTryingMove AND bFirstCycle THEN
	eEntranceState[1].bCapPutted := TRUE;
	eEntranceState[1].bCapOK:= FALSE;
	eEntranceState[1].bFormPresent := TRUE; // jeżeli zanik czujnik formatki i nie było formatki to wpisz ze nie było butelki
END_IF
//JEZELI WLACZONO SPRAWDZANIE FORMATEK Z TRIGERCOUNTER TO
IF bWithFormControlTrigerCounter  AND bTriggerCounter AND NOT bKeepTryingMove AND bFirstCycle THEN
	eEntranceState[1].bFormPresent := TRUE;
END_IF



//PRZESUNIECIE
IF (*iEntranceArrayElements <= iExitArrayElements AND*) bFirstCycle  THEN
		IF rtbTrigger.Q OR bKeepTryingMove OR bTriggerCounter THEN
		bTriggerCounter := FALSE; 
		bKeepTryingMove := FALSE;
		nFormCounter := 0;
		bBottlePresent := bCapPresent  := FALSE; 
		FOR i:= 1 TO iExitArrayElements-1 DO // SORTOWANIE
			IF NOT eExitState[i].bFormPresent THEN 
				eExitState[i] := eExitState[i+1];
				eExitState[i+1] := eClearPackageState;
			END_IF
		END_FOR

		FOR i := 1 TO iExitArrayElements DO
			IF  NOT eExitState[i].bFormPresent THEN  		// Jeżeli w rejestrze wyjściowym jest wolne miejsce to wpisz rejestr wejściowy
				
			
				eExitState[i]	:=	eEntranceState[1];			// Wpisz do rejestru dane np z [1] Buffor do [1,2,3,4,5,6] Package
				eEntranceState[1]	:=	eClearPackageState;		// Czyszczenie pierwszego rejestru wejściowego			
				k:=i;	

									// Przepisywanie zmiennej pomocniczej
				FOR i := 1 TO iEntranceArrayElements DO   				
					IF i = iEntranceArrayElements THEN
						eEntranceState[i]:=eClearPackageState;			// Zerowanie ostatniego bo zostało przesuniete wszystko o 1
					ELSE												// Przepisanie 2 do 1, 3 do 2, 4 do 3, 5 do 4, 6 do 5, zeruj 6
						eEntranceState[i] := eEntranceState[i+1]; 		// 2 do 1, 3 do 2,
						eEntranceState[i+1]:= eClearPackageState;		// zeruj 2, 
						iLFTest2:=iLFTest2;
					END_IF
				END_FOR
				
				
				
				
				bTriggerDone := TRUE;
				EXIT;
				bError := TRUE;
				iError := 5;
			ELSE
				nFormCounter := nFormCounter + 1;
				bError := TRUE;
				iError := 6;
			END_IF
		END_FOR

		IF nFormCounter = iExitArrayElements THEN
			bKeepTryingMove:=NOT bNoKeepTryingMove;
		END_IF
	END_IF
END_IF


//CZYSZCZENIE REJESTRU WEJSCIOWEGO
IF rtbReset.Q THEN
	FOR r1 := 1 TO iEntranceArrayElements DO
		eEntranceState[r1] := eClearPackageState;
	END_FOR
	FOR r2 := 1 TO iExitArrayElements DO
		eExitState[r2] := eClearPackageState;
	END_FOR
	bKeepTryingMove :=FALSE;
	bTriggerDone := FALSE;
	bTriggerCounter := FALSE; 
	nFormCounter := 0;
	bBottlePresent := bCapPresent := FALSE; 
	bError := FALSE;
	iError := 0;
END_IF

END_FUNCTION_BLOCK

// ---- POUs/FB/FB_MoveRegisterLF.TcPOU
(*
Nazwa:			FB_MoveRegister
Opis:			Blok przesuniecia rejestru formatek
Wersja:			v0.3 		
Data:			2018-11-16
Autor:			DP
Urzadzenia:		 
Konfiguracja:	
Info:
- Są dwa rejestry, wejściowy i wyjsciowy (struktury)
- Jezeli rejestr ma np. 6 elementów to za kazdym razem po wykryciu trigera program będzie
	1 wejściowy przesuwał na 1 wolny (nie ma formatki) wyjściowy
	kasował 1 rejestr wejściowy
	przesuwal rejetr wejsciowy 2 na 1(przeniesiony i skasowany), 3 na 2, 4 na 3, 5 na 4, 6 na 5 i kasowal 6wejsciowy
	tym sposobem po 6 trigerach caly rejestr wejsciowy powinien być na wyjsciowym
	np po 3 trigerach na wyjsciowym powinny byc zajete 1 do 3 i na wejsciowym 1 do 3
Błędy:
1 - nie wyszło z pętli for
2 - formatka już jest w rejestrze
Uwagi:
- 
Zmiany:
2018-09-18 Dodano sprawdzanie nasadek
2018-06-14 DP Pierwsza wersja
*)

FUNCTION_BLOCK FB_MoveRegisterLF
VAR_INPUT
	bFirstCycle:BOOL;					//Pierwszy cykl, zeby na początku nie wykrywało zbocza opadającego
	bTrigger :BOOL;						// Przesuniecie tablicy o jeden
	tTriggerFilterTimeOn:TIME:=T#0MS;	// Czas filtrowania wejścia Trigger na załączenie
	tTriggerFilterTimeOff:TIME:=T#0MS;	// Czas filtrowania wejścia Trigger na wyłączenie
	bTriggerBottle :BOOL;				// Zapisywanie czy jest butelka czy nie (jezeli kontrola wlączona)
	bWithBottleControl: BOOL;			// Włączona opcja kontroli butelek
	bWithCapControl:BOOL;				// Wlaczona kontrola nasadek
	bWithFormControlTrigerCounter:BOOL;	// Jezeku na trigercontrol nie ma formatki do przesunięcia to stwórz nową
	bMoveOnlyToLastExitRegister:BOOL;	// Przepisuj rejestr wejściowy tylko na ostatni wyjściowy bez przesunięcia wyjściowego
	bMoveOnlyIfFormPresent:BOOL;		// Przepisuj tylko jak jest formatka
	bRotateEntranceRegisterBefore:BOOL;	// Najpierw przesuń rejestr wejściowy a następnie z niego zabierz
	bNoKeepTryingMove:BOOL;				// Dalej przepisuj jezeli nie ma miejsca
	bTriggerCap: BOOL;					// Truger wykrycia nasadki
	bReset :BOOL;						// Czyszczenie tablic
	iEntranceArrayElements :UINT; 		// Wartość koncowa tablicy
	iExitArrayElements :UINT; 			// Wartość koncowa tablicy
	bInvertWriting :BOOL;				// Wpisywanie odwrotne zamist z 1entrance na 1exit to 1entrance na 6exit	
	eClearPackageState :S_PackageState; // Czysty rejestr
END_VAR
VAR_IN_OUT
	bTriggerCounter :BOOL;		// Triger ktory jest kasowany
	eEntranceState :ARRAY [1..17] OF S_PackageState;	
	eExitState :ARRAY [1..17] OF S_PackageState;
	bKeepTryingMove :BOOL;		// Probuj dalej zapisać formatki aż się któraś zwolni
END_VAR

VAR_OUTPUT	
	bError :BOOL; 				// Błąd
	iError: UINT;				// Nr Błędu
	bTriggerDone :BOOL; 		// Wykonano przesunięcie
	bTriggerFilteredOUT:BOOL;	//Wyjscie przefiltrowanego sygnalu wejsciowego
END_VAR

VAR
	i:UINT;						// Zmienna w tablicy
	k:UINT;						// Pomocnicza zmienna do zapisywnia czy jest butelka
	rtbTrigger :R_TRIG;			// Reaguje na zbocze
	rtbTriggerBottle :R_TRIG;	// Reaguje na zbocze
	rtbReset :R_TRIG;			// Reaguje na zbocze
	TimerResetErrors :TON;		// Reset Błedu
	nFormCounter :UINT;					//Licznik formatek
	r1,r2:UINT;
	bBottlePresent: BOOL;				//Zmienna pomocnicza ze wykryto butelkę
	bCapPresent: BOOL;					//Zmienna pomocnicza ze wykryto butelkę
	j: UINT;
	tonTriggerFilterTimeOn: TON;
	bTriggerFiltered: BOOL;
	tofTriggerFilterTimeOff: TOF;
	tonTriggerFilterTimeBeforeTrigger: TON;
END_VAR

//Filtrowanie sygnału wejściowego
tofTriggerFilterTimeOff	(IN:=bTrigger, PT:=tTriggerFilterTimeOff);
tonTriggerFilterTimeOn	(IN:=tofTriggerFilterTimeOff.Q, PT:=tTriggerFilterTimeOn);
bTriggerFiltered 		:= tonTriggerFilterTimeOn.Q;
bTriggerFilteredOUT		:= bTriggerFiltered ;

//TRIGI I TIMERY
IF bWithBottleControl THEN
	rtbTrigger 	(CLK := NOT bTriggerFiltered, Q=>);
	rtbTriggerBottle 	(CLK := NOT bTriggerBottle, Q=>);
ELSIF bWithCapControl THEN
	rtbTrigger 	(CLK := NOT bTriggerFiltered, Q=>);
ELSE
	rtbTrigger 	(CLK := bTriggerFiltered, Q=>);
	rtbTriggerBottle 	(CLK := bTriggerBottle, Q=>);
END_IF

rtbReset 	(CLK := bReset, Q=>);
TimerResetErrors (IN:= bError, PT:=T#1000MS, Q=>);

//RESETOWANIE BLEDU
IF TimerResetErrors.Q THEN
	bError := FALSE;
END_IF

//KASOWANIE ZMIENNYCH
bTriggerDone := FALSE;

//JEZELI WLACZONO KONTROLE BUTELEK TO NADPISUJ REJESTR CZY JEST BUTELKA
IF bWithBottleControl AND bTrigger AND bTriggerBottle AND NOT bKeepTryingMove THEN //Jezeli od wykrycia formatki liczy TIMER i wykryło butelke to wpisz do rejestru że jest butelka
	eEntranceState[1].bBottlePresent := TRUE;
	eEntranceState[1].bFormPresent := TRUE;
	bBottlePresent := TRUE; // Wpisuje że jest butelka jezeli wystąpi sygnał podczas trwania czujnika formatki
ELSIF bWithBottleControl AND rtbTrigger.Q AND NOT bBottlePresent AND  NOT bKeepTryingMove AND bFirstCycle THEN
	eEntranceState[1].bBottlePresent := FALSE;
	eEntranceState[1].bFormPresent := TRUE; // jeżeli zanik czujnik formatki i nie było formatki to wpisz ze nie było butelki
END_IF
//JEZELI WLACZONO KONTROLE NASADEk TO NADPISUJ REJESTR CZY JEST BUTELKA 
(*IF bWithCapControl AND bTrigger AND bTriggerCap AND NOT bKeepTryingMove THEN //Jezeli od wykrycia formatki liczy TIMER i wykryło butelke to wpisz do rejestru że jest butelka
	eEntranceState[1].bCapPutted := TRUE;
	eEntranceState[1].bCapOK := TRUE; eEntranceState[1].bBottlePresent:= TRUE;//Zmiana nowa
	eEntranceState[1].bFormPresent := TRUE;
	bCapPresent := TRUE; // Wpisuje że jest butelka jezeli wystąpi sygnał podczas trwania czujnika formatki*)
	//ZMIANA LU 192
IF bWithCapControl AND bTriggerCap AND NOT bKeepTryingMove THEN //Jezeli od wykrycia formatki liczy TIMER i wykryło butelke to wpisz do rejestru że jest butelka
	eEntranceState[1].bCapPutted := TRUE;
	eEntranceState[1].bCapOK := TRUE; eEntranceState[1].bBottlePresent:= TRUE;//Zmiana nowa
	eEntranceState[1].bFormPresent := TRUE;
	bCapPresent := TRUE; // Wpisuje że jest butelka jezeli wystąpi sygnał podczas trwania czujnika formatki	
ELSIF bWithCapControl AND rtbTrigger.Q AND NOT bCapPresent AND  NOT bKeepTryingMove AND bFirstCycle THEN
	eEntranceState[1].bCapPutted := TRUE;
	eEntranceState[1].bCapOK:= FALSE;
	eEntranceState[1].bFormPresent := TRUE; // jeżeli zanik czujnik formatki i nie było formatki to wpisz ze nie było butelki
END_IF
//JEZELI WLACZONO SPRAWDZANIE FORMATEK Z TRIGERCOUNTER TO
IF bWithFormControlTrigerCounter  AND (bTriggerCounter OR rtbTrigger.Q) AND NOT bKeepTryingMove AND bFirstCycle THEN //Zmiena UBL50, tworz tez nowa jak Trigger
	eEntranceState[1].bFormPresent := TRUE;
END_IF

